LIN {X 0,Y 418.247,Z 151.387,A -85,B 0,C 180,E1 -10284.852,E2 -10284.852} C_VEL
LIN {X 0,Y 418.21,Z 151.394,A -85,B 0,C 180,E1 -10288.069,E2 -10288.069} C_VEL
LIN {X 0,Y 418.241,Z 151.389,A -85,B 0,C 180,E1 -10291.019,E2 -10291.019} C_VEL
LIN {X 0,Y 418.237,Z 151.391,A -85,B 0,C 180,E1 -10293.678,E2 -10293.678} C_VEL
LIN {X 0,Y 418.28,Z 151.466,A -85,B 0,C 180,E1 -10294.622,E2 -10294.622} C_VEL
LIN {X 0,Y 420.263,Z 161.531,A -85,B 0,C 180,E1 -10297.015,E2 -10297.015} C_VEL
LIN {X 0,Y 420.369,Z 166.895,A -85,B 0,C 180,E1 -10298.213,E2 -10298.213} C_VEL
LIN {X 0,Y 420.18,Z 169.806,A -85,B 0,C 180,E1 -10298.846,E2 -10298.846} C_VEL
LIN {X 0,Y 424.258,Z 189.635,A -85,B 0,C 180,E1 -10299.44,E2 -10299.44} C_VEL
LIN {X 0,Y 423.077,Z 277.594,A -85,B 0,C 180,E1 -10301.015,E2 -10301.015} C_VEL
LIN {X 0,Y 422.644,Z 290.834,A -85,B 0,C 180,E1 -10301.445,E2 -10301.445} C_VEL
LIN {X 0,Y 422.214,Z 302.953,A -85,B 0,C 180,E1 -10302.028,E2 -10302.028} C_VEL
LIN {X 0,Y 421.492,Z 314.996,A -85,B 0,C 180,E1 -10302.805,E2 -10302.805} C_VEL
LIN {X 0,Y 420.748,Z 326.21,A -85,B 0,C 180,E1 -10303.744,E2 -10303.744} C_VEL
LIN {X 0,Y 420.06,Z 336.204,A -85,B 0,C 180,E1 -10304.788,E2 -10304.788} C_VEL
LIN {X 0,Y 419.384,Z 345.484,A -85,B 0,C 180,E1 -10305.977,E2 -10305.977} C_VEL
LIN {X 0,Y 418.655,Z 354.531,A -85,B 0,C 180,E1 -10307.422,E2 -10307.422} C_VEL
LIN {X 0,Y 418.062,Z 362.564,A -85,B 0,C 180,E1 -10309.032,E2 -10309.032} C_VEL
LIN {X 0,Y 417.595,Z 369.077,A -85,B 0,C 180,E1 -10310.73,E2 -10310.73} C_VEL
LIN {X 0,Y 417.327,Z 373.741,A -85,B 0,C 180,E1 -10312.327,E2 -10312.327} C_VEL
LIN {X 0,Y 417.08,Z 377.245,A -85,B 0,C 180,E1 -10313.982,E2 -10313.982} C_VEL
LIN {X 0,Y 416.893,Z 379.545,A -85,B 0,C 180,E1 -10315.695,E2 -10315.695} C_VEL
LIN {X 0,Y 416.841,Z 380.55,A -85,B 0,C 180,E1 -10317.46,E2 -10317.46} C_VEL
LIN {X 0,Y 416.876,Z 380.209,A -85,B 0,C 180,E1 -10319.294,E2 -10319.294} C_VEL
LIN {X 0,Y 416.992,Z 378.31,A -85,B 0,C 180,E1 -10321.213,E2 -10321.213} C_VEL
LIN {X 0,Y 417.215,Z 375.163,A -85,B 0,C 180,E1 -10322.947,E2 -10322.947} C_VEL
LIN {X 0,Y 417.47,Z 370.897,A -85,B 0,C 180,E1 -10324.577,E2 -10324.577} C_VEL
LIN {X 0,Y 417.714,Z 365.312,A -85,B 0,C 180,E1 -10326.184,E2 -10326.184} C_VEL
LIN {X 0,Y 418.151,Z 359.125,A -85,B 0,C 180,E1 -10327.579,E2 -10327.579} C_VEL
LIN {X 0,Y 418.736,Z 350.665,A -85,B 0,C 180,E1 -10329.105,E2 -10329.105} C_VEL
LIN {X 0,Y 419.408,Z 341.621,A -85,B 0,C 180,E1 -10330.419,E2 -10330.419} C_VEL
LIN {X 0,Y 420.06,Z 331.76,A -85,B 0,C 180,E1 -10331.575,E2 -10331.575} C_VEL
LIN {X 0,Y 420.835,Z 320.491,A -85,B 0,C 180,E1 -10332.631,E2 -10332.631} C_VEL
LIN {X 0,Y 421.361,Z 310.208,A -85,B 0,C 180,E1 -10333.403,E2 -10333.403} C_VEL
LIN {X 0,Y 421.938,Z 298.072,A -85,B 0,C 180,E1 -10334.11,E2 -10334.11} C_VEL
LIN {X 0,Y 422.395,Z 285.579,A -85,B 0,C 180,E1 -10334.628,E2 -10334.628} C_VEL
LIN {X 0,Y 422.729,Z 272.036,A -85,B 0,C 180,E1 -10334.985,E2 -10334.985} C_VEL
LIN {X 0,Y 423.075,Z 245.782,A -85,B 0,C 180,E1 -10335.443,E2 -10335.443} C_VEL
LIN {X 0,Y 422.465,Z 239.979,A -85,B 0,C 180,E1 -10335.571,E2 -10335.571} C_VEL
LIN {X 0,Y 417.244,Z 221.285,A -85,B 0,C 180,E1 -10336.126,E2 -10336.126} C_VEL
LIN {X 0,Y 416.667,Z 215.482,A -85,B 0,C 180,E1 -10336.257,E2 -10336.257} C_VEL
LIN {X 0,Y 416.96,Z 190.299,A -85,B 0,C 180,E1 -10336.708,E2 -10336.708} C_VEL
LIN {X 0,Y 412.975,Z 169.781,A -85,B 0,C 180,E1 -10337.281,E2 -10337.281} C_VEL
LIN {X 0,Y 413.217,Z 162.427,A -85,B 0,C 180,E1 -10338.969,E2 -10338.969} C_VEL
LIN {X 0,Y 411.366,Z 152.245,A -85,B 0,C 180,E1 -10341.495,E2 -10341.495} C_VEL
LIN {X 0,Y 411.435,Z 152.237,A -85,B 0,C 180,E1 -10344.117,E2 -10344.117} C_VEL
LIN {X 0,Y 411.511,Z 152.224,A -85,B 0,C 180,E1 -10348.043,E2 -10348.043} C_VEL
LIN {X 0,Y 411.439,Z 152.231,A -85,B 0,C 180,E1 -10350.979,E2 -10350.979} C_VEL
LIN {X 0,Y 411.433,Z 152.232,A -85,B 0,C 180,E1 -10352.937,E2 -10352.937} C_VEL
LIN {X 0,Y 411.432,Z 152.234,A -85,B 0,C 180,E1 -10355.883,E2 -10355.883} C_VEL
LIN {X 0,Y 411.319,Z 152.246,A -85,B 0,C 180,E1 -10358.846,E2 -10358.846} C_VEL
LIN {X 0,Y 411.285,Z 152.254,A -85,B 0,C 180,E1 -10361.833,E2 -10361.833} C_VEL
LIN {X 0,Y 411.234,Z 152.256,A -85,B 0,C 180,E1 -10364.854,E2 -10364.854} C_VEL
LIN {X 0,Y 411.232,Z 152.263,A -85,B 0,C 180,E1 -10367.916,E2 -10367.916} C_VEL
LIN {X 0,Y 411.199,Z 152.26,A -85,B 0,C 180,E1 -10371.034,E2 -10371.034} C_VEL
LIN {X 0,Y 411.194,Z 152.263,A -85,B 0,C 180,E1 -10374.218,E2 -10374.218} C_VEL
LIN {X 0,Y 411.174,Z 152.268,A -85,B 0,C 180,E1 -10377.484,E2 -10377.484} C_VEL
LIN {X 0,Y 411.199,Z 152.267,A -85,B 0,C 180,E1 -10379.713,E2 -10379.713} C_VEL
LIN {X 0,Y 411.207,Z 152.262,A -85,B 0,C 180,E1 -10383.156,E2 -10383.156} C_VEL
LIN {X 0,Y 411.194,Z 152.261,A -85,B 0,C 180,E1 -10386.552,E2 -10386.552} C_VEL
LIN {X 0,Y 411.172,Z 152.267,A -85,B 0,C 180,E1 -10389.72,E2 -10389.72} C_VEL
LIN {X 0,Y 411.165,Z 152.269,A -85,B 0,C 180,E1 -10393.135,E2 -10393.135} C_VEL
LIN {X 0,Y 411.166,Z 152.265,A -85,B 0,C 180,E1 -10395.882,E2 -10395.882} C_VEL
LIN {X 0,Y 411.165,Z 152.268,A -85,B 0,C 180,E1 -10399.494,E2 -10399.494} C_VEL
LIN {X 0,Y 411.19,Z 152.261,A -85,B 0,C 180,E1 -10402.026,E2 -10402.026} C_VEL
LIN {X 0,Y 411.196,Z 152.262,A -85,B 0,C 180,E1 -10405.665,E2 -10405.665} C_VEL
LIN {X 0,Y 411.19,Z 152.266,A -85,B 0,C 180,E1 -10409.152,E2 -10409.152} C_VEL
LIN {X 0,Y 411.181,Z 152.264,A -85,B 0,C 180,E1 -10411.407,E2 -10411.407} C_VEL
LIN {X 0,Y 411.215,Z 152.264,A -85,B 0,C 180,E1 -10414.934,E2 -10414.934} C_VEL
LIN {X 0,Y 411.206,Z 152.26,A -85,B 0,C 180,E1 -10417.913,E2 -10417.913} C_VEL
LIN {X 0,Y 411.218,Z 152.261,A -85,B 0,C 180,E1 -10421.051,E2 -10421.051} C_VEL
LIN {X 0,Y 411.213,Z 152.261,A -85,B 0,C 180,E1 -10424.13,E2 -10424.13} C_VEL
LIN {X 0,Y 411.307,Z 152.248,A -85,B 0,C 180,E1 -10427.166,E2 -10427.166} C_VEL
LIN {X 0,Y 411.289,Z 152.253,A -85,B 0,C 180,E1 -10430.161,E2 -10430.161} C_VEL
LIN {X 0,Y 411.394,Z 152.236,A -85,B 0,C 180,E1 -10433.132,E2 -10433.132} C_VEL
LIN {X 0,Y 411.292,Z 152.249,A -85,B 0,C 180,E1 -10435.099,E2 -10435.099} C_VEL
LIN {X 0,Y 411.506,Z 152.227,A -85,B 0,C 180,E1 -10438.042,E2 -10438.042} C_VEL
LIN {X 0,Y 411.381,Z 152.238,A -85,B 0,C 180,E1 -10440.979,E2 -10440.979} C_VEL
LIN {X 0,Y 411.43,Z 152.232,A -85,B 0,C 180,E1 -10442.937,E2 -10442.937} C_VEL
LIN {X 0,Y 411.394,Z 152.236,A -85,B 0,C 180,E1 -10446.868,E2 -10446.868} C_VEL
LIN {X 0,Y 411.279,Z 152.256,A -85,B 0,C 180,E1 -10449.839,E2 -10449.839} C_VEL
LIN {X 0,Y 411.303,Z 152.248,A -85,B 0,C 180,E1 -10453.1,E2 -10453.1} C_VEL
LIN {X 0,Y 411.208,Z 152.259,A -85,B 0,C 180,E1 -10456.891,E2 -10456.891} C_VEL
LIN {X 0,Y 411.205,Z 152.263,A -85,B 0,C 180,E1 -10459.988,E2 -10459.988} C_VEL
LIN {X 0,Y 411.187,Z 152.264,A -85,B 0,C 180,E1 -10463.149,E2 -10463.149} C_VEL
LIN {X 0,Y 411.166,Z 152.265,A -85,B 0,C 180,E1 -10466.386,E2 -10466.386} C_VEL
LIN {X 0,Y 411.194,Z 152.265,A -85,B 0,C 180,E1 -10469.713,E2 -10469.713} C_VEL
LIN {X 0,Y 411.205,Z 152.264,A -85,B 0,C 180,E1 -10473.156,E2 -10473.156} C_VEL
LIN {X 0,Y 411.19,Z 152.262,A -85,B 0,C 180,E1 -10476.551,E2 -10476.551} C_VEL
LIN {X 0,Y 411.169,Z 152.266,A -85,B 0,C 180,E1 -10479.72,E2 -10479.72} C_VEL
LIN {X 0,Y 411.163,Z 152.272,A -85,B 0,C 180,E1 -10483.135,E2 -10483.135} C_VEL
LIN {X 0,Y 411.165,Z 152.265,A -85,B 0,C 180,E1 -10485.882,E2 -10485.882} C_VEL
LIN {X 0,Y 411.159,Z 152.267,A -85,B 0,C 180,E1 -10489.493,E2 -10489.493} C_VEL
LIN {X 0,Y 411.181,Z 152.263,A -85,B 0,C 180,E1 -10492.024,E2 -10492.024} C_VEL
LIN {X 0,Y 411.201,Z 152.264,A -85,B 0,C 180,E1 -10495.124,E2 -10495.124} C_VEL
LIN {X 0,Y 411.155,Z 152.266,A -85,B 0,C 180,E1 -10498.001,E2 -10498.001} C_VEL
LIN {X 0,Y 411.168,Z 152.269,A -85,B 0,C 180,E1 -10501.406,E2 -10501.406} C_VEL
LIN {X 0,Y 411.195,Z 152.457,A -85,B 0,C 180,E1 -10502.596,E2 -10502.596} C_VEL
LIN {X 0,Y 413.73,Z 164.949,A -85,B 0,C 180,E1 -10505.406,E2 -10505.406} C_VEL
LIN {X 0,Y 414.147,Z 168.979,A -85,B 0,C 180,E1 -10506.272,E2 -10506.272} C_VEL
LIN {X 0,Y 413.042,Z 185.931,A -85,B 0,C 180,E1 -10509.723,E2 -10509.723} C_VEL
LIN {X 0,Y 412.619,Z 190.946,A -85,B 0,C 180,E1 -10510.731,E2 -10510.731} C_VEL
LIN {X 0,Y 416.688,Z 217.687,A -85,B 0,C 180,E1 -10511.42,E2 -10511.42} C_VEL
LIN {X 0,Y 415.709,Z 299.077,A -85,B 0,C 180,E1 -10512.886,E2 -10512.886} C_VEL
LIN {X 0,Y 415.217,Z 312.276,A -85,B 0,C 180,E1 -10513.309,E2 -10513.309} C_VEL
LIN {X 0,Y 414.543,Z 325.557,A -85,B 0,C 180,E1 -10513.945,E2 -10513.945} C_VEL
LIN {X 0,Y 413.796,Z 337.523,A -85,B 0,C 180,E1 -10514.737,E2 -10514.737} C_VEL
LIN {X 0,Y 413.007,Z 349.008,A -85,B 0,C 180,E1 -10515.716,E2 -10515.716} C_VEL
LIN {X 0,Y 412.314,Z 359.362,A -85,B 0,C 180,E1 -10516.822,E2 -10516.822} C_VEL
LIN {X 0,Y 411.736,Z 367.828,A -85,B 0,C 180,E1 -10517.93,E2 -10517.93} C_VEL
LIN {X 0,Y 410.994,Z 376.995,A -85,B 0,C 180,E1 -10519.407,E2 -10519.407} C_VEL
LIN {X 0,Y 410.556,Z 384.382,A -85,B 0,C 180,E1 -10520.889,E2 -10520.889} C_VEL
LIN {X 0,Y 410.287,Z 389.386,A -85,B 0,C 180,E1 -10522.124,E2 -10522.124} C_VEL
LIN {X 0,Y 410.043,Z 394.737,A -85,B 0,C 180,E1 -10523.775,E2 -10523.775} C_VEL
LIN {X 0,Y 410.016,Z 397.958,A -85,B 0,C 180,E1 -10525.083,E2 -10525.083} C_VEL
LIN {X 0,Y 409.931,Z 399.873,A -85,B 0,C 180,E1 -10526.068,E2 -10526.068} C_VEL
LIN {X 0,Y 409.926,Z 401.342,A -85,B 0,C 180,E1 -10527.052,E2 -10527.052} C_VEL
LIN {X 0,Y 409.967,Z 402.374,A -85,B 0,C 180,E1 -10528.035,E2 -10528.035} C_VEL
LIN {X 0,Y 409.936,Z 403.011,A -85,B 0,C 180,E1 -10529.018,E2 -10529.018} C_VEL
LIN {X 0,Y 409.928,Z 403.258,A -85,B 0,C 180,E1 -10530,E2 -10530} C_VEL
LIN {X 0,Y 409.936,Z 403.087,A -85,B 0,C 180,E1 -10530.982,E2 -10530.982} C_VEL
LIN {X 0,Y 409.967,Z 402.495,A -85,B 0,C 180,E1 -10531.965,E2 -10531.965} C_VEL
LIN {X 0,Y 409.931,Z 400.127,A -85,B 0,C 180,E1 -10533.932,E2 -10533.932} C_VEL
LIN {X 0,Y 410.012,Z 397.209,A -85,B 0,C 180,E1 -10535.41,E2 -10535.41} C_VEL
LIN {X 0,Y 410.166,Z 393.255,A -85,B 0,C 180,E1 -10536.889,E2 -10536.889} C_VEL
LIN {X 0,Y 410.419,Z 388.163,A -85,B 0,C 180,E1 -10538.369,E2 -10538.369} C_VEL
LIN {X 0,Y 410.807,Z 381.768,A -85,B 0,C 180,E1 -10539.851,E2 -10539.851} C_VEL
LIN {X 0,Y 411.366,Z 373.767,A -85,B 0,C 180,E1 -10541.331,E2 -10541.331} C_VEL
LIN {X 0,Y 412.105,Z 365.627,A -85,B 0,C 180,E1 -10542.559,E2 -10542.559} C_VEL
LIN {X 0,Y 412.797,Z 355.709,A -85,B 0,C 180,E1 -10543.79,E2 -10543.79} C_VEL
LIN {X 0,Y 413.618,Z 344.608,A -85,B 0,C 180,E1 -10544.892,E2 -10544.892} C_VEL
LIN {X 0,Y 414.356,Z 333.75,A -85,B 0,C 180,E1 -10545.747,E2 -10545.747} C_VEL
LIN {X 0,Y 415.195,Z 321.802,A -85,B 0,C 180,E1 -10546.471,E2 -10546.471} C_VEL
LIN {X 0,Y 415.792,Z 308.86,A -85,B 0,C 180,E1 -10547.047,E2 -10547.047} C_VEL
LIN {X 0,Y 416.332,Z 296.141,A -85,B 0,C 180,E1 -10547.404,E2 -10547.404} C_VEL
LIN {X 0,Y 417.271,Z 216.994,A -85,B 0,C 180,E1 -10548.837,E2 -10548.837} C_VEL
LIN {X 0,Y 413.255,Z 192.477,A -85,B 0,C 180,E1 -10549.503,E2 -10549.503} C_VEL
LIN {X 0,Y 412.87,Z 190.246,A -85,B 0,C 180,E1 -10549.585,E2 -10549.585} C_VEL
LIN {X 0,Y 413.986,Z 173.404,A -85,B 0,C 180,E1 -10552.983,E2 -10552.983} C_VEL
LIN {X 0,Y 414.341,Z 168.316,A -85,B 0,C 180,E1 -10554.022,E2 -10554.022} C_VEL
LIN {X 0,Y 412.433,Z 158.109,A -85,B 0,C 180,E1 -10556.299,E2 -10556.299} C_VEL
LIN {X 0,Y 411.162,Z 152.272,A -85,B 0,C 180,E1 -10557.692,E2 -10557.692} C_VEL
LIN {X 0,Y 411.183,Z 152.269,A -85,B 0,C 180,E1 -10560.848,E2 -10560.848} C_VEL
LIN {X 0,Y 411.19,Z 152.267,A -85,B 0,C 180,E1 -10564.335,E2 -10564.335} C_VEL
LIN {X 0,Y 411.185,Z 152.266,A -85,B 0,C 180,E1 -10566.743,E2 -10566.743} C_VEL
LIN {X 0,Y 411.164,Z 152.269,A -85,B 0,C 180,E1 -10569.719,E2 -10569.719} C_VEL
LIN {X 0,Y 411.162,Z 152.274,A -85,B 0,C 180,E1 -10573.136,E2 -10573.136} C_VEL
LIN {X 0,Y 411.165,Z 152.268,A -85,B 0,C 180,E1 -10575.882,E2 -10575.882} C_VEL
LIN {X 0,Y 411.158,Z 152.265,A -85,B 0,C 180,E1 -10579.493,E2 -10579.493} C_VEL
LIN {X 0,Y 411.179,Z 152.265,A -85,B 0,C 180,E1 -10582.024,E2 -10582.024} C_VEL
LIN {X 0,Y 411.202,Z 152.264,A -85,B 0,C 180,E1 -10585.124,E2 -10585.124} C_VEL
LIN {X 0,Y 411.156,Z 152.265,A -85,B 0,C 180,E1 -10588.002,E2 -10588.002} C_VEL
LIN {X 0,Y 411.17,Z 152.262,A -85,B 0,C 180,E1 -10591.406,E2 -10591.406} C_VEL
LIN {X 0,Y 411.19,Z 152.259,A -85,B 0,C 180,E1 -10594.942,E2 -10594.942} C_VEL
LIN {X 0,Y 411.199,Z 152.262,A -85,B 0,C 180,E1 -10597.913,E2 -10597.913} C_VEL
LIN {X 0,Y 411.182,Z 152.265,A -85,B 0,C 180,E1 -10601.049,E2 -10601.049} C_VEL
LIN {X 0,Y 411.199,Z 152.259,A -85,B 0,C 180,E1 -10604.129,E2 -10604.129} C_VEL
LIN {X 0,Y 411.299,Z 152.248,A -85,B 0,C 180,E1 -10607.166,E2 -10607.166} C_VEL
LIN {X 0,Y 411.277,Z 152.25,A -85,B 0,C 180,E1 -10610.161,E2 -10610.161} C_VEL
LIN {X 0,Y 411.392,Z 152.23,A -85,B 0,C 180,E1 -10613.132,E2 -10613.132} C_VEL
LIN {X 0,Y 411.286,Z 152.249,A -85,B 0,C 180,E1 -10615.099,E2 -10615.099} C_VEL
LIN {X 0,Y 411.506,Z 152.22,A -85,B 0,C 180,E1 -10618.043,E2 -10618.043} C_VEL
LIN {X 0,Y 411.381,Z 152.236,A -85,B 0,C 180,E1 -10620.979,E2 -10620.979} C_VEL
LIN {X 0,Y 411.43,Z 152.232,A -85,B 0,C 180,E1 -10622.938,E2 -10622.938} C_VEL
LIN {X 0,Y 411.394,Z 152.237,A -85,B 0,C 180,E1 -10626.868,E2 -10626.868} C_VEL
LIN {X 0,Y 411.28,Z 152.252,A -85,B 0,C 180,E1 -10629.839,E2 -10629.839} C_VEL
LIN {X 0,Y 411.309,Z 152.246,A -85,B 0,C 180,E1 -10633.103,E2 -10633.103} C_VEL
LIN {X 0,Y 411.211,Z 152.261,A -85,B 0,C 180,E1 -10636.891,E2 -10636.891} C_VEL
LIN {X 0,Y 411.207,Z 152.263,A -85,B 0,C 180,E1 -10639.988,E2 -10639.988} C_VEL
LIN {X 0,Y 411.192,Z 152.265,A -85,B 0,C 180,E1 -10643.148,E2 -10643.148} C_VEL
LIN {X 0,Y 411.178,Z 152.269,A -85,B 0,C 180,E1 -10646.385,E2 -10646.385} C_VEL
LIN {X 0,Y 411.198,Z 152.267,A -85,B 0,C 180,E1 -10649.713,E2 -10649.713} C_VEL
LIN {X 0,Y 411.208,Z 152.265,A -85,B 0,C 180,E1 -10653.156,E2 -10653.156} C_VEL
LIN {X 0,Y 411.217,Z 152.351,A -85,B 0,C 180,E1 -10654.333,E2 -10654.333} C_VEL
LIN {X 0,Y 413.378,Z 163.207,A -85,B 0,C 180,E1 -10656.958,E2 -10656.958} C_VEL
LIN {X 0,Y 413.45,Z 168.137,A -85,B 0,C 180,E1 -10658.077,E2 -10658.077} C_VEL
LIN {X 0,Y 413.332,Z 170.075,A -85,B 0,C 180,E1 -10658.506,E2 -10658.506} C_VEL
LIN {X 0,Y 417.683,Z 191.349,A -85,B 0,C 180,E1 -10659.142,E2 -10659.142} C_VEL
LIN {X 0,Y 416.348,Z 277.624,A -85,B 0,C 180,E1 -10660.707,E2 -10660.707} C_VEL
LIN {X 0,Y 415.892,Z 291.111,A -85,B 0,C 180,E1 -10661.151,E2 -10661.151} C_VEL
LIN {X 0,Y 415.423,Z 303.31,A -85,B 0,C 180,E1 -10661.749,E2 -10661.749} C_VEL
LIN {X 0,Y 414.653,Z 315.611,A -85,B 0,C 180,E1 -10662.563,E2 -10662.563} C_VEL
LIN {X 0,Y 413.844,Z 327.228,A -85,B 0,C 180,E1 -10663.564,E2 -10663.564} C_VEL
LIN {X 0,Y 413.044,Z 337.978,A -85,B 0,C 180,E1 -10664.733,E2 -10664.733} C_VEL
LIN {X 0,Y 412.299,Z 347.356,A -85,B 0,C 180,E1 -10666.009,E2 -10666.009} C_VEL
LIN {X 0,Y 411.681,Z 354.747,A -85,B 0,C 180,E1 -10667.229,E2 -10667.229} C_VEL
LIN {X 0,Y 411.07,Z 362.421,A -85,B 0,C 180,E1 -10668.787,E2 -10668.787} C_VEL
LIN {X 0,Y 410.601,Z 368.581,A -85,B 0,C 180,E1 -10670.375,E2 -10670.375} C_VEL
LIN {X 0,Y 410.279,Z 373.398,A -85,B 0,C 180,E1 -10671.997,E2 -10671.997} C_VEL
LIN {X 0,Y 410.033,Z 377.03,A -85,B 0,C 180,E1 -10673.667,E2 -10673.667} C_VEL
LIN {X 0,Y 409.804,Z 379.64,A -85,B 0,C 180,E1 -10675.532,E2 -10675.532} C_VEL
LIN {X 0,Y 409.739,Z 380.707,A -85,B 0,C 180,E1 -10677.19,E2 -10677.19} C_VEL
LIN {X 0,Y 409.765,Z 380.532,A -85,B 0,C 180,E1 -10679.045,E2 -10679.045} C_VEL
LIN {X 0,Y 409.829,Z 379.751,A -85,B 0,C 180,E1 -10680.178,E2 -10680.178} C_VEL
LIN {X 0,Y 409.903,Z 378.415,A -85,B 0,C 180,E1 -10681.309,E2 -10681.309} C_VEL
LIN {X 0,Y 410.129,Z 375.365,A -85,B 0,C 180,E1 -10683.009,E2 -10683.009} C_VEL
LIN {X 0,Y 410.41,Z 371.144,A -85,B 0,C 180,E1 -10684.652,E2 -10684.652} C_VEL
LIN {X 0,Y 410.677,Z 365.574,A -85,B 0,C 180,E1 -10686.286,E2 -10686.286} C_VEL
LIN {X 0,Y 411.18,Z 358.374,A -85,B 0,C 180,E1 -10687.912,E2 -10687.912} C_VEL
LIN {X 0,Y 411.795,Z 349.969,A -85,B 0,C 180,E1 -10689.421,E2 -10689.421} C_VEL
LIN {X 0,Y 412.499,Z 340.937,A -85,B 0,C 180,E1 -10690.725,E2 -10690.725} C_VEL
LIN {X 0,Y 413.23,Z 330.683,A -85,B 0,C 180,E1 -10691.917,E2 -10691.917} C_VEL
LIN {X 0,Y 414.005,Z 319.36,A -85,B 0,C 180,E1 -10692.972,E2 -10692.972} C_VEL
LIN {X 0,Y 414.639,Z 307.674,A -85,B 0,C 180,E1 -10693.823,E2 -10693.823} C_VEL
LIN {X 0,Y 415.16,Z 295.909,A -85,B 0,C 180,E1 -10694.473,E2 -10694.473} C_VEL
LIN {X 0,Y 415.664,Z 282.878,A -85,B 0,C 180,E1 -10694.984,E2 -10694.984} C_VEL
LIN {X 0,Y 415.96,Z 269.747,A -85,B 0,C 180,E1 -10695.297,E2 -10695.297} C_VEL
LIN {X 0,Y 416.667,Z 215.482,A -85,B 0,C 180,E1 -10696.257,E2 -10696.257} C_VEL
LIN {X 0,Y 416.139,Z 209.665,A -85,B 0,C 180,E1 -10696.387,E2 -10696.387} C_VEL
LIN {X 0,Y 413.596,Z 200.312,A -85,B 0,C 180,E1 -10696.671,E2 -10696.671} C_VEL
LIN {X 0,Y 411.065,Z 192.914,A -85,B 0,C 180,E1 -10696.922,E2 -10696.922} C_VEL
LIN {X 0,Y 409.064,Z 185.346,A -85,B 0,C 180,E1 -10697.155,E2 -10697.155} C_VEL
LIN {X 0,Y 406.073,Z 169.943,A -85,B 0,C 180,E1 -10697.601,E2 -10697.601} C_VEL
LIN {X 0,Y 406.261,Z 163.82,A -85,B 0,C 180,E1 -10699.03,E2 -10699.03} C_VEL
LIN {X 0,Y 404.318,Z 153.123,A -85,B 0,C 180,E1 -10701.724,E2 -10701.724} C_VEL
LIN {X 0,Y 404.382,Z 153.116,A -85,B 0,C 180,E1 -10704.014,E2 -10704.014} C_VEL
LIN {X 0,Y 404.48,Z 153.1,A -85,B 0,C 180,E1 -10708.008,E2 -10708.008} C_VEL
LIN {X 0,Y 404.404,Z 153.108,A -85,B 0,C 180,E1 -10710.996,E2 -10710.996} C_VEL
LIN {X 0,Y 404.392,Z 153.109,A -85,B 0,C 180,E1 -10712.989,E2 -10712.989} C_VEL
LIN {X 0,Y 404.38,Z 153.114,A -85,B 0,C 180,E1 -10715.986,E2 -10715.986} C_VEL
LIN {X 0,Y 404.267,Z 153.124,A -85,B 0,C 180,E1 -10719.002,E2 -10719.002} C_VEL
LIN {X 0,Y 404.258,Z 153.132,A -85,B 0,C 180,E1 -10722.042,E2 -10722.042} C_VEL
LIN {X 0,Y 404.179,Z 153.135,A -85,B 0,C 180,E1 -10725.119,E2 -10725.119} C_VEL
LIN {X 0,Y 404.196,Z 153.136,A -85,B 0,C 180,E1 -10728.239,E2 -10728.239} C_VEL
LIN {X 0,Y 404.141,Z 153.142,A -85,B 0,C 180,E1 -10731.419,E2 -10731.419} C_VEL
LIN {X 0,Y 404.15,Z 153.138,A -85,B 0,C 180,E1 -10734.668,E2 -10734.668} C_VEL
LIN {X 0,Y 404.118,Z 153.146,A -85,B 0,C 180,E1 -10738.006,E2 -10738.006} C_VEL
LIN {X 0,Y 404.146,Z 153.14,A -85,B 0,C 180,E1 -10740.285,E2 -10740.285} C_VEL
LIN {X 0,Y 404.14,Z 153.144,A -85,B 0,C 180,E1 -10743.813,E2 -10743.813} C_VEL
LIN {X 0,Y 404.137,Z 153.141,A -85,B 0,C 180,E1 -10746.875,E2 -10746.875} C_VEL
LIN {X 0,Y 404.119,Z 153.143,A -85,B 0,C 180,E1 -10750.075,E2 -10750.075} C_VEL
LIN {X 0,Y 404.144,Z 153.143,A -85,B 0,C 180,E1 -10753.082,E2 -10753.082} C_VEL
LIN {X 0,Y 404.123,Z 153.143,A -85,B 0,C 180,E1 -10755.922,E2 -10755.922} C_VEL
LIN {X 0,Y 404.106,Z 153.145,A -85,B 0,C 180,E1 -10758.633,E2 -10758.633} C_VEL
LIN {X 0,Y 404.145,Z 153.142,A -85,B 0,C 180,E1 -10761.494,E2 -10761.494} C_VEL
LIN {X 0,Y 404.177,Z 153.141,A -85,B 0,C 180,E1 -10764.983,E2 -10764.983} C_VEL
LIN {X 0,Y 404.14,Z 153.141,A -85,B 0,C 180,E1 -10768.443,E2 -10768.443} C_VEL
LIN {X 0,Y 404.154,Z 153.145,A -85,B 0,C 180,E1 -10770.863,E2 -10770.863} C_VEL
LIN {X 0,Y 404.143,Z 153.141,A -85,B 0,C 180,E1 -10774.231,E2 -10774.231} C_VEL
LIN {X 0,Y 404.169,Z 153.136,A -85,B 0,C 180,E1 -10777.508,E2 -10777.508} C_VEL
LIN {X 0,Y 404.163,Z 153.143,A -85,B 0,C 180,E1 -10780.707,E2 -10780.707} C_VEL
LIN {X 0,Y 404.184,Z 153.135,A -85,B 0,C 180,E1 -10783.846,E2 -10783.846} C_VEL
LIN {X 0,Y 404.287,Z 153.124,A -85,B 0,C 180,E1 -10786.939,E2 -10786.939} C_VEL
LIN {X 0,Y 404.256,Z 153.128,A -85,B 0,C 180,E1 -10789.988,E2 -10789.988} C_VEL
LIN {X 0,Y 404.344,Z 153.115,A -85,B 0,C 180,E1 -10793.012,E2 -10793.012} C_VEL
LIN {X 0,Y 404.263,Z 153.125,A -85,B 0,C 180,E1 -10795.013,E2 -10795.013} C_VEL
LIN {X 0,Y 404.475,Z 153.102,A -85,B 0,C 180,E1 -10798.008,E2 -10798.008} C_VEL
LIN {X 0,Y 404.352,Z 153.114,A -85,B 0,C 180,E1 -10800.996,E2 -10800.996} C_VEL
LIN {X 0,Y 404.389,Z 153.109,A -85,B 0,C 180,E1 -10802.989,E2 -10802.989} C_VEL
LIN {X 0,Y 404.37,Z 153.117,A -85,B 0,C 180,E1 -10805.986,E2 -10805.986} C_VEL
LIN {X 0,Y 404.259,Z 153.125,A -85,B 0,C 180,E1 -10809.002,E2 -10809.002} C_VEL
LIN {X 0,Y 404.249,Z 153.131,A -85,B 0,C 180,E1 -10812.042,E2 -10812.042} C_VEL
LIN {X 0,Y 404.16,Z 153.138,A -85,B 0,C 180,E1 -10815.12,E2 -10815.12} C_VEL
LIN {X 0,Y 404.13,Z 153.143,A -85,B 0,C 180,E1 -10818.242,E2 -10818.242} C_VEL
LIN {X 0,Y 404.129,Z 153.145,A -85,B 0,C 180,E1 -10821.42,E2 -10821.42} C_VEL
LIN {X 0,Y 404.136,Z 153.14,A -85,B 0,C 180,E1 -10824.668,E2 -10824.668} C_VEL
LIN {X 0,Y 404.101,Z 153.146,A -85,B 0,C 180,E1 -10828.007,E2 -10828.007} C_VEL
LIN {X 0,Y 404.141,Z 153.14,A -85,B 0,C 180,E1 -10830.286,E2 -10830.286} C_VEL
LIN {X 0,Y 404.138,Z 153.142,A -85,B 0,C 180,E1 -10833.813,E2 -10833.813} C_VEL
LIN {X 0,Y 404.133,Z 153.143,A -85,B 0,C 180,E1 -10836.874,E2 -10836.874} C_VEL
LIN {X 0,Y 404.119,Z 153.142,A -85,B 0,C 180,E1 -10840.075,E2 -10840.075} C_VEL
LIN {X 0,Y 404.143,Z 153.146,A -85,B 0,C 180,E1 -10843.082,E2 -10843.082} C_VEL
LIN {X 0,Y 404.122,Z 153.142,A -85,B 0,C 180,E1 -10845.922,E2 -10845.922} C_VEL
LIN {X 0,Y 404.102,Z 153.147,A -85,B 0,C 180,E1 -10848.632,E2 -10848.632} C_VEL
LIN {X 0,Y 404.138,Z 153.141,A -85,B 0,C 180,E1 -10851.495,E2 -10851.495} C_VEL
LIN {X 0,Y 404.172,Z 153.141,A -85,B 0,C 180,E1 -10854.982,E2 -10854.982} C_VEL
LIN {X 0,Y 404.132,Z 153.144,A -85,B 0,C 180,E1 -10858.444,E2 -10858.444} C_VEL
LIN {X 0,Y 404.148,Z 153.145,A -85,B 0,C 180,E1 -10860.862,E2 -10860.862} C_VEL
LIN {X 0,Y 404.169,Z 153.289,A -85,B 0,C 180,E1 -10862.333,E2 -10862.333} C_VEL
LIN {X 0,Y 406.703,Z 165.919,A -85,B 0,C 180,E1 -10865.225,E2 -10865.225} C_VEL
LIN {X 0,Y 407.202,Z 170.22,A -85,B 0,C 180,E1 -10866.169,E2 -10866.169} C_VEL
LIN {X 0,Y 406.019,Z 187.492,A -85,B 0,C 180,E1 -10869.745,E2 -10869.745} C_VEL
LIN {X 0,Y 405.704,Z 190.807,A -85,B 0,C 180,E1 -10870.422,E2 -10870.422} C_VEL
LIN {X 0,Y 409.925,Z 218.175,A -85,B 0,C 180,E1 -10871.133,E2 -10871.133} C_VEL
LIN {X 0,Y 408.886,Z 299.259,A -85,B 0,C 180,E1 -10872.624,E2 -10872.624} C_VEL
LIN {X 0,Y 408.343,Z 313.089,A -85,B 0,C 180,E1 -10873.084,E2 -10873.084} C_VEL
LIN {X 0,Y 407.649,Z 326.057,A -85,B 0,C 180,E1 -10873.73,E2 -10873.73} C_VEL
LIN {X 0,Y 406.817,Z 338.65,A -85,B 0,C 180,E1 -10874.597,E2 -10874.597} C_VEL
LIN {X 0,Y 406.032,Z 349.897,A -85,B 0,C 180,E1 -10875.593,E2 -10875.593} C_VEL
LIN {X 0,Y 405.268,Z 360.185,A -85,B 0,C 180,E1 -10876.739,E2 -10876.739} C_VEL
LIN {X 0,Y 404.621,Z 369.147,A -85,B 0,C 180,E1 -10877.969,E2 -10877.969} C_VEL
LIN {X 0,Y 403.905,Z 378.058,A -85,B 0,C 180,E1 -10879.473,E2 -10879.473} C_VEL
LIN {X 0,Y 403.473,Z 385.201,A -85,B 0,C 180,E1 -10880.981,E2 -10880.981} C_VEL
LIN {X 0,Y 403.137,Z 390.89,A -85,B 0,C 180,E1 -10882.487,E2 -10882.487} C_VEL
LIN {X 0,Y 402.938,Z 395.363,A -85,B 0,C 180,E1 -10883.993,E2 -10883.993} C_VEL
LIN {X 0,Y 402.928,Z 397.723,A -85,B 0,C 180,E1 -10884.997,E2 -10884.997} C_VEL
LIN {X 0,Y 402.851,Z 399.646,A -85,B 0,C 180,E1 -10885.998,E2 -10885.998} C_VEL
LIN {X 0,Y 402.825,Z 401.127,A -85,B 0,C 180,E1 -10887,E2 -10887} C_VEL
LIN {X 0,Y 402.865,Z 402.165,A -85,B 0,C 180,E1 -10888.001,E2 -10888.001} C_VEL
LIN {X 0,Y 402.863,Z 402.808,A -85,B 0,C 180,E1 -10889,E2 -10889} C_VEL
LIN {X 0,Y 402.853,Z 403.061,A -85,B 0,C 180,E1 -10890,E2 -10890} C_VEL
LIN {X 0,Y 402.863,Z 402.9,A -85,B 0,C 180,E1 -10891,E2 -10891} C_VEL
LIN {X 0,Y 402.864,Z 402.312,A -85,B 0,C 180,E1 -10892,E2 -10892} C_VEL
LIN {X 0,Y 402.851,Z 399.953,A -85,B 0,C 180,E1 -10894.002,E2 -10894.002} C_VEL
LIN {X 0,Y 402.909,Z 397.044,A -85,B 0,C 180,E1 -10895.505,E2 -10895.505} C_VEL
LIN {X 0,Y 403.08,Z 393.098,A -85,B 0,C 180,E1 -10897.011,E2 -10897.011} C_VEL
LIN {X 0,Y 403.36,Z 388.016,A -85,B 0,C 180,E1 -10898.517,E2 -10898.517} C_VEL
LIN {X 0,Y 403.802,Z 381.643,A -85,B 0,C 180,E1 -10900.023,E2 -10900.023} C_VEL
LIN {X 0,Y 404.385,Z 373.668,A -85,B 0,C 180,E1 -10901.529,E2 -10901.529} C_VEL
LIN {X 0,Y 405.159,Z 365.557,A -85,B 0,C 180,E1 -10902.778,E2 -10902.778} C_VEL
LIN {X 0,Y 405.873,Z 355.673,A -85,B 0,C 180,E1 -10904.03,E2 -10904.03} C_VEL
LIN {X 0,Y 406.764,Z 344.626,A -85,B 0,C 180,E1 -10905.149,E2 -10905.149} C_VEL
LIN {X 0,Y 407.539,Z 333.819,A -85,B 0,C 180,E1 -10906.017,E2 -10906.017} C_VEL
LIN {X 0,Y 408.412,Z 321.946,A -85,B 0,C 180,E1 -10906.753,E2 -10906.753} C_VEL
LIN {X 0,Y 409.037,Z 309.184,A -85,B 0,C 180,E1 -10907.338,E2 -10907.338} C_VEL
LIN {X 0,Y 409.602,Z 295.396,A -85,B 0,C 180,E1 -10907.732,E2 -10907.732} C_VEL
LIN {X 0,Y 410.506,Z 216.867,A -85,B 0,C 180,E1 -10909.182,E2 -10909.182} C_VEL
LIN {X 0,Y 406.354,Z 192.13,A -85,B 0,C 180,E1 -10909.88,E2 -10909.88} C_VEL
LIN {X 0,Y 406.022,Z 190,A -85,B 0,C 180,E1 -10909.964,E2 -10909.964} C_VEL
LIN {X 0,Y 407.356,Z 171.699,A -85,B 0,C 180,E1 -10913.727,E2 -10913.727} C_VEL
LIN {X 0,Y 407.24,Z 168.248,A -85,B 0,C 180,E1 -10914.468,E2 -10914.468} C_VEL
LIN {X 0,Y 405.197,Z 158.058,A -85,B 0,C 180,E1 -10916.806,E2 -10916.806} C_VEL
LIN {X 0,Y 404.118,Z 153.152,A -85,B 0,C 180,E1 -10918.006,E2 -10918.006} C_VEL
LIN {X 0,Y 404.14,Z 153.148,A -85,B 0,C 180,E1 -10920.286,E2 -10920.286} C_VEL
LIN {X 0,Y 404.137,Z 153.147,A -85,B 0,C 180,E1 -10923.813,E2 -10923.813} C_VEL
LIN {X 0,Y 404.131,Z 153.145,A -85,B 0,C 180,E1 -10926.874,E2 -10926.874} C_VEL
LIN {X 0,Y 404.119,Z 153.146,A -85,B 0,C 180,E1 -10930.075,E2 -10930.075} C_VEL
LIN {X 0,Y 404.142,Z 153.149,A -85,B 0,C 180,E1 -10933.082,E2 -10933.082} C_VEL
LIN {X 0,Y 404.122,Z 153.145,A -85,B 0,C 180,E1 -10935.922,E2 -10935.922} C_VEL
LIN {X 0,Y 404.102,Z 153.15,A -85,B 0,C 180,E1 -10938.633,E2 -10938.633} C_VEL
LIN {X 0,Y 404.135,Z 153.143,A -85,B 0,C 180,E1 -10941.496,E2 -10941.496} C_VEL
LIN {X 0,Y 404.173,Z 153.141,A -85,B 0,C 180,E1 -10944.983,E2 -10944.983} C_VEL
LIN {X 0,Y 404.133,Z 153.143,A -85,B 0,C 180,E1 -10948.444,E2 -10948.444} C_VEL
LIN {X 0,Y 404.149,Z 153.137,A -85,B 0,C 180,E1 -10950.862,E2 -10950.862} C_VEL
LIN {X 0,Y 404.154,Z 153.136,A -85,B 0,C 180,E1 -10954.724,E2 -10954.724} C_VEL
LIN {X 0,Y 404.165,Z 153.137,A -85,B 0,C 180,E1 -10957.508,E2 -10957.508} C_VEL
LIN {X 0,Y 404.135,Z 153.143,A -85,B 0,C 180,E1 -10960.706,E2 -10960.706} C_VEL
LIN {X 0,Y 404.174,Z 153.134,A -85,B 0,C 180,E1 -10963.846,E2 -10963.846} C_VEL
LIN {X 0,Y 404.268,Z 153.125,A -85,B 0,C 180,E1 -10966.938,E2 -10966.938} C_VEL
LIN {X 0,Y 404.245,Z 153.124,A -85,B 0,C 180,E1 -10969.988,E2 -10969.988} C_VEL
LIN {X 0,Y 404.342,Z 153.108,A -85,B 0,C 180,E1 -10973.012,E2 -10973.012} C_VEL
LIN {X 0,Y 404.258,Z 153.124,A -85,B 0,C 180,E1 -10975.013,E2 -10975.013} C_VEL
LIN {X 0,Y 404.474,Z 153.095,A -85,B 0,C 180,E1 -10978.009,E2 -10978.009} C_VEL
LIN {X 0,Y 404.351,Z 153.111,A -85,B 0,C 180,E1 -10980.996,E2 -10980.996} C_VEL
LIN {X 0,Y 404.363,Z 153.112,A -85,B 0,C 180,E1 -10982.989,E2 -10982.989} C_VEL
LIN {X 0,Y 404.342,Z 153.113,A -85,B 0,C 180,E1 -10986.485,E2 -10986.485} C_VEL
LIN {X 0,Y 404.26,Z 153.123,A -85,B 0,C 180,E1 -10989.002,E2 -10989.002} C_VEL
LIN {X 0,Y 404.253,Z 153.128,A -85,B 0,C 180,E1 -10992.042,E2 -10992.042} C_VEL
LIN {X 0,Y 404.178,Z 153.137,A -85,B 0,C 180,E1 -10995.119,E2 -10995.119} C_VEL
LIN {X 0,Y 404.139,Z 153.143,A -85,B 0,C 180,E1 -10998.242,E2 -10998.242} C_VEL
LIN {X 0,Y 404.135,Z 153.145,A -85,B 0,C 180,E1 -11001.42,E2 -11001.42} C_VEL
LIN {X 0,Y 404.152,Z 153.143,A -85,B 0,C 180,E1 -11004.667,E2 -11004.667} C_VEL
LIN {X 0,Y 404.106,Z 153.152,A -85,B 0,C 180,E1 -11008.007,E2 -11008.007} C_VEL
LIN {X 0,Y 404.145,Z 153.144,A -85,B 0,C 180,E1 -11010.285,E2 -11010.285} C_VEL
LIN {X 0,Y 404.201,Z 153.279,A -85,B 0,C 180,E1 -11014.032,E2 -11014.032} C_VEL
LIN {X 0,Y 406.319,Z 163.813,A -85,B 0,C 180,E1 -11016.637,E2 -11016.637} C_VEL
LIN {X 0,Y 406.662,Z 166.791,A -85,B 0,C 180,E1 -11017.346,E2 -11017.346} C_VEL
LIN {X 0,Y 406.5,Z 170.434,A -85,B 0,C 180,E1 -11018.145,E2 -11018.145} C_VEL
LIN {X 0,Y 410.928,Z 191.578,A -85,B 0,C 180,E1 -11018.797,E2 -11018.797} C_VEL
LIN {X 0,Y 409.607,Z 278.396,A -85,B 0,C 180,E1 -11020.409,E2 -11020.409} C_VEL
LIN {X 0,Y 409.136,Z 292.217,A -85,B 0,C 180,E1 -11020.883,E2 -11020.883} C_VEL
LIN {X 0,Y 408.573,Z 305.291,A -85,B 0,C 180,E1 -11021.56,E2 -11021.56} C_VEL
LIN {X 0,Y 407.725,Z 317.522,A -85,B 0,C 180,E1 -11022.413,E2 -11022.413} C_VEL
LIN {X 0,Y 406.992,Z 327.769,A -85,B 0,C 180,E1 -11023.329,E2 -11023.329} C_VEL
LIN {X 0,Y 406.169,Z 337.981,A -85,B 0,C 180,E1 -11024.458,E2 -11024.458} C_VEL
LIN {X 0,Y 405.379,Z 347.513,A -85,B 0,C 180,E1 -11025.773,E2 -11025.773} C_VEL
LIN {X 0,Y 404.547,Z 356.71,A -85,B 0,C 180,E1 -11027.349,E2 -11027.349} C_VEL
LIN {X 0,Y 403.951,Z 364.022,A -85,B 0,C 180,E1 -11028.945,E2 -11028.945} C_VEL
LIN {X 0,Y 403.495,Z 369.931,A -85,B 0,C 180,E1 -11030.585,E2 -11030.585} C_VEL
LIN {X 0,Y 403.153,Z 374.88,A -85,B 0,C 180,E1 -11032.4,E2 -11032.4} C_VEL
LIN {X 0,Y 402.962,Z 377.326,A -85,B 0,C 180,E1 -11033.63,E2 -11033.63} C_VEL
LIN {X 0,Y 402.741,Z 379.427,A -85,B 0,C 180,E1 -11035.102,E2 -11035.102} C_VEL
LIN {X 0,Y 402.663,Z 380.797,A -85,B 0,C 180,E1 -11036.907,E2 -11036.907} C_VEL
LIN {X 0,Y 402.648,Z 380.852,A -85,B 0,C 180,E1 -11038.79,E2 -11038.79} C_VEL
LIN {X 0,Y 402.768,Z 379.359,A -85,B 0,C 180,E1 -11040.752,E2 -11040.752} C_VEL
LIN {X 0,Y 402.868,Z 377.798,A -85,B 0,C 180,E1 -11041.9,E2 -11041.9} C_VEL
LIN {X 0,Y 403.143,Z 374.377,A -85,B 0,C 180,E1 -11043.606,E2 -11043.606} C_VEL
LIN {X 0,Y 403.414,Z 369.69,A -85,B 0,C 180,E1 -11045.284,E2 -11045.284} C_VEL
LIN {X 0,Y 403.781,Z 363.924,A -85,B 0,C 180,E1 -11046.869,E2 -11046.869} C_VEL
LIN {X 0,Y 404.234,Z 357.316,A -85,B 0,C 180,E1 -11048.318,E2 -11048.318} C_VEL
LIN {X 0,Y 404.874,Z 349.638,A -85,B 0,C 180,E1 -11049.685,E2 -11049.685} C_VEL
LIN {X 0,Y 405.605,Z 340.215,A -85,B 0,C 180,E1 -11051.041,E2 -11051.041} C_VEL
LIN {X 0,Y 406.331,Z 330.28,A -85,B 0,C 180,E1 -11052.2,E2 -11052.2} C_VEL
LIN {X 0,Y 407.1,Z 319.751,A -85,B 0,C 180,E1 -11053.192,E2 -11053.192} C_VEL
LIN {X 0,Y 407.792,Z 307.683,A -85,B 0,C 180,E1 -11054.084,E2 -11054.084} C_VEL
LIN {X 0,Y 408.356,Z 295.077,A -85,B 0,C 180,E1 -11054.783,E2 -11054.783} C_VEL
LIN {X 0,Y 408.873,Z 282.217,A -85,B 0,C 180,E1 -11055.281,E2 -11055.281} C_VEL
LIN {X 0,Y 409.175,Z 267.79,A -85,B 0,C 180,E1 -11055.61,E2 -11055.61} C_VEL
LIN {X 0,Y 410.217,Z 191.382,A -85,B 0,C 180,E1 -11056.989,E2 -11056.989} C_VEL
LIN {X 0,Y 409.064,Z 185.346,A -85,B 0,C 180,E1 -11057.155,E2 -11057.155} C_VEL
LIN {X 0,Y 407.507,Z 180.011,A -85,B 0,C 180,E1 -11057.381,E2 -11057.381} C_VEL
LIN {X 0,Y 405.281,Z 175.244,A -85,B 0,C 180,E1 -11057.733,E2 -11057.733} C_VEL
LIN {X 0,Y 402.087,Z 169.715,A -85,B 0,C 180,E1 -11058.371,E2 -11058.371} C_VEL
LIN {X 0,Y 400.068,Z 166.114,A -85,B 0,C 180,E1 -11058.966,E2 -11058.966} C_VEL
LIN {X 0,Y 398.903,Z 162.979,A -85,B 0,C 180,E1 -11059.652,E2 -11059.652} C_VEL
LIN {X 0,Y 397.299,Z 153.995,A -85,B 0,C 180,E1 -11061.964,E2 -11061.964} C_VEL
LIN {X 0,Y 397.242,Z 154.001,A -85,B 0,C 180,E1 -11064.925,E2 -11064.925} C_VEL
LIN {X 0,Y 397.449,Z 153.975,A -85,B 0,C 180,E1 -11067.973,E2 -11067.973} C_VEL
LIN {X 0,Y 397.369,Z 153.984,A -85,B 0,C 180,E1 -11071.013,E2 -11071.013} C_VEL
LIN {X 0,Y 397.327,Z 153.989,A -85,B 0,C 180,E1 -11073.042,E2 -11073.042} C_VEL
LIN {X 0,Y 397.331,Z 153.993,A -85,B 0,C 180,E1 -11076.092,E2 -11076.092} C_VEL
LIN {X 0,Y 397.237,Z 154,A -85,B 0,C 180,E1 -11079.162,E2 -11079.162} C_VEL
LIN {X 0,Y 397.221,Z 154.006,A -85,B 0,C 180,E1 -11082.258,E2 -11082.258} C_VEL
LIN {X 0,Y 397.127,Z 154.014,A -85,B 0,C 180,E1 -11085.394,E2 -11085.394} C_VEL
LIN {X 0,Y 397.153,Z 154.011,A -85,B 0,C 180,E1 -11088.574,E2 -11088.574} C_VEL
LIN {X 0,Y 397.098,Z 154.024,A -85,B 0,C 180,E1 -11091.819,E2 -11091.819} C_VEL
LIN {X 0,Y 397.098,Z 154.018,A -85,B 0,C 180,E1 -11095.136,E2 -11095.136} C_VEL
LIN {X 0,Y 397.072,Z 154.02,A -85,B 0,C 180,E1 -11098.548,E2 -11098.548} C_VEL
LIN {X 0,Y 397.083,Z 154.023,A -85,B 0,C 180,E1 -11101.836,E2 -11101.836} C_VEL
LIN {X 0,Y 397.122,Z 154.014,A -85,B 0,C 180,E1 -11104.494,E2 -11104.494} C_VEL
LIN {X 0,Y 397.095,Z 154.018,A -85,B 0,C 180,E1 -11108.276,E2 -11108.276} C_VEL
LIN {X 0,Y 397.054,Z 154.023,A -85,B 0,C 180,E1 -11111.977,E2 -11111.977} C_VEL
LIN {X 0,Y 397.088,Z 154.023,A -85,B 0,C 180,E1 -11115.069,E2 -11115.069} C_VEL
LIN {X 0,Y 397.054,Z 154.023,A -85,B 0,C 180,E1 -11118.024,E2 -11118.024} C_VEL
LIN {X 0,Y 397.096,Z 154.018,A -85,B 0,C 180,E1 -11121.724,E2 -11121.724} C_VEL
LIN {X 0,Y 397.12,Z 154.016,A -85,B 0,C 180,E1 -11125.506,E2 -11125.506} C_VEL
LIN {X 0,Y 397.079,Z 154.024,A -85,B 0,C 180,E1 -11129.117,E2 -11129.117} C_VEL
LIN {X 0,Y 397.094,Z 154.021,A -85,B 0,C 180,E1 -11132.602,E2 -11132.602} C_VEL
LIN {X 0,Y 397.115,Z 154.015,A -85,B 0,C 180,E1 -11135.98,E2 -11135.98} C_VEL
LIN {X 0,Y 397.142,Z 154.011,A -85,B 0,C 180,E1 -11139.705,E2 -11139.705} C_VEL
LIN {X 0,Y 397.157,Z 154.014,A -85,B 0,C 180,E1 -11142.859,E2 -11142.859} C_VEL
LIN {X 0,Y 397.233,Z 154.005,A -85,B 0,C 180,E1 -11146.703,E2 -11146.703} C_VEL
LIN {X 0,Y 397.216,Z 154.003,A -85,B 0,C 180,E1 -11149.809,E2 -11149.809} C_VEL
LIN {X 0,Y 397.297,Z 153.994,A -85,B 0,C 180,E1 -11152.887,E2 -11152.887} C_VEL
LIN {X 0,Y 397.235,Z 154.001,A -85,B 0,C 180,E1 -11154.925,E2 -11154.925} C_VEL
LIN {X 0,Y 397.443,Z 153.978,A -85,B 0,C 180,E1 -11157.973,E2 -11157.973} C_VEL
LIN {X 0,Y 397.443,Z 153.98,A -85,B 0,C 180,E1 -11162.027,E2 -11162.027} C_VEL
LIN {X 0,Y 397.323,Z 153.995,A -85,B 0,C 180,E1 -11166.092,E2 -11166.092} C_VEL
LIN {X 0,Y 397.23,Z 154.001,A -85,B 0,C 180,E1 -11169.162,E2 -11169.162} C_VEL
LIN {X 0,Y 397.211,Z 154.006,A -85,B 0,C 180,E1 -11172.258,E2 -11172.258} C_VEL
LIN {X 0,Y 397.112,Z 154.018,A -85,B 0,C 180,E1 -11175.395,E2 -11175.395} C_VEL
LIN {X 0,Y 397.085,Z 154.019,A -85,B 0,C 180,E1 -11178.577,E2 -11178.577} C_VEL
LIN {X 0,Y 397.09,Z 154.023,A -85,B 0,C 180,E1 -11181.819,E2 -11181.819} C_VEL
LIN {X 0,Y 397.104,Z 154.018,A -85,B 0,C 180,E1 -11185.135,E2 -11185.135} C_VEL
LIN {X 0,Y 397.062,Z 154.021,A -85,B 0,C 180,E1 -11188.548,E2 -11188.548} C_VEL
LIN {X 0,Y 397.077,Z 154.022,A -85,B 0,C 180,E1 -11191.834,E2 -11191.834} C_VEL
LIN {X 0,Y 397.117,Z 154.015,A -85,B 0,C 180,E1 -11194.494,E2 -11194.494} C_VEL
LIN {X 0,Y 397.091,Z 154.018,A -85,B 0,C 180,E1 -11198.277,E2 -11198.277} C_VEL
LIN {X 0,Y 397.053,Z 154.023,A -85,B 0,C 180,E1 -11201.976,E2 -11201.976} C_VEL
LIN {X 0,Y 397.088,Z 154.025,A -85,B 0,C 180,E1 -11205.069,E2 -11205.069} C_VEL
LIN {X 0,Y 397.052,Z 154.023,A -85,B 0,C 180,E1 -11208.024,E2 -11208.024} C_VEL
LIN {X 0,Y 397.09,Z 154.018,A -85,B 0,C 180,E1 -11211.723,E2 -11211.723} C_VEL
LIN {X 0,Y 397.116,Z 154.015,A -85,B 0,C 180,E1 -11215.505,E2 -11215.505} C_VEL
LIN {X 0,Y 397.072,Z 154.025,A -85,B 0,C 180,E1 -11219.117,E2 -11219.117} C_VEL
LIN {X 0,Y 397.097,Z 154.155,A -85,B 0,C 180,E1 -11222.066,E2 -11222.066} C_VEL
LIN {X 0,Y 399.693,Z 166.873,A -85,B 0,C 180,E1 -11225.039,E2 -11225.039} C_VEL
LIN {X 0,Y 400.168,Z 171.987,A -85,B 0,C 180,E1 -11226.175,E2 -11226.175} C_VEL
LIN {X 0,Y 399.013,Z 188.456,A -85,B 0,C 180,E1 -11229.643,E2 -11229.643} C_VEL
LIN {X 0,Y 398.839,Z 190.841,A -85,B 0,C 180,E1 -11230.104,E2 -11230.104} C_VEL
LIN {X 0,Y 403.148,Z 219.393,A -85,B 0,C 180,E1 -11230.855,E2 -11230.855} C_VEL
LIN {X 0,Y 402.072,Z 299.25,A -85,B 0,C 180,E1 -11232.352,E2 -11232.352} C_VEL
LIN {X 0,Y 401.502,Z 313.019,A -85,B 0,C 180,E1 -11232.819,E2 -11232.819} C_VEL
LIN {X 0,Y 400.824,Z 325.437,A -85,B 0,C 180,E1 -11233.445,E2 -11233.445} C_VEL
LIN {X 0,Y 400.022,Z 336.542,A -85,B 0,C 180,E1 -11234.197,E2 -11234.197} C_VEL
LIN {X 0,Y 399.186,Z 348.139,A -85,B 0,C 180,E1 -11235.209,E2 -11235.209} C_VEL
LIN {X 0,Y 398.46,Z 358.328,A -85,B 0,C 180,E1 -11236.323,E2 -11236.323} C_VEL
LIN {X 0,Y 397.801,Z 367.137,A -85,B 0,C 180,E1 -11237.501,E2 -11237.501} C_VEL
LIN {X 0,Y 396.961,Z 376.376,A -85,B 0,C 180,E1 -11239.028,E2 -11239.028} C_VEL
LIN {X 0,Y 396.469,Z 383.81,A -85,B 0,C 180,E1 -11240.563,E2 -11240.563} C_VEL
LIN {X 0,Y 396.174,Z 388.854,A -85,B 0,C 180,E1 -11241.841,E2 -11241.841} C_VEL
LIN {X 0,Y 395.919,Z 393.742,A -85,B 0,C 180,E1 -11243.375,E2 -11243.375} C_VEL
LIN {X 0,Y 395.84,Z 397.489,A -85,B 0,C 180,E1 -11244.907,E2 -11244.907} C_VEL
LIN {X 0,Y 395.774,Z 399.419,A -85,B 0,C 180,E1 -11245.927,E2 -11245.927} C_VEL
LIN {X 0,Y 395.728,Z 400.912,A -85,B 0,C 180,E1 -11246.946,E2 -11246.946} C_VEL
LIN {X 0,Y 395.763,Z 401.956,A -85,B 0,C 180,E1 -11247.965,E2 -11247.965} C_VEL
LIN {X 0,Y 395.792,Z 402.606,A -85,B 0,C 180,E1 -11248.983,E2 -11248.983} C_VEL
LIN {X 0,Y 395.78,Z 402.863,A -85,B 0,C 180,E1 -11250,E2 -11250} C_VEL
LIN {X 0,Y 395.792,Z 402.713,A -85,B 0,C 180,E1 -11251.017,E2 -11251.017} C_VEL
LIN {X 0,Y 395.762,Z 402.129,A -85,B 0,C 180,E1 -11252.035,E2 -11252.035} C_VEL
LIN {X 0,Y 395.774,Z 399.783,A -85,B 0,C 180,E1 -11254.073,E2 -11254.073} C_VEL
LIN {X 0,Y 395.824,Z 396.458,A -85,B 0,C 180,E1 -11255.801,E2 -11255.801} C_VEL
LIN {X 0,Y 396.072,Z 391.391,A -85,B 0,C 180,E1 -11257.648,E2 -11257.648} C_VEL
LIN {X 0,Y 396.504,Z 384.889,A -85,B 0,C 180,E1 -11259.437,E2 -11259.437} C_VEL
LIN {X 0,Y 397.033,Z 377.782,A -85,B 0,C 180,E1 -11260.97,E2 -11260.97} C_VEL
LIN {X 0,Y 397.897,Z 368.914,A -85,B 0,C 180,E1 -11262.496,E2 -11262.496} C_VEL
LIN {X 0,Y 398.592,Z 360.129,A -85,B 0,C 180,E1 -11263.732,E2 -11263.732} C_VEL
LIN {X 0,Y 399.448,Z 350.22,A -85,B 0,C 180,E1 -11264.872,E2 -11264.872} C_VEL
LIN {X 0,Y 400.38,Z 338.784,A -85,B 0,C 180,E1 -11265.919,E2 -11265.919} C_VEL
LIN {X 0,Y 401.289,Z 326.406,A -85,B 0,C 180,E1 -11266.797,E2 -11266.797} C_VEL
LIN {X 0,Y 402.005,Z 314.688,A -85,B 0,C 180,E1 -11267.421,E2 -11267.421} C_VEL
LIN {X 0,Y 402.658,Z 302.107,A -85,B 0,C 180,E1 -11267.884,E2 -11267.884} C_VEL
LIN {X 0,Y 403.05,Z 284.725,A -85,B 0,C 180,E1 -11268.26,E2 -11268.26} C_VEL
LIN {X 0,Y 403.875,Z 218.007,A -85,B 0,C 180,E1 -11269.509,E2 -11269.509} C_VEL
LIN {X 0,Y 399.922,Z 194.118,A -85,B 0,C 180,E1 -11270.2,E2 -11270.2} C_VEL
LIN {X 0,Y 399.143,Z 189.76,A -85,B 0,C 180,E1 -11270.36,E2 -11270.36} C_VEL
LIN {X 0,Y 400.509,Z 171.683,A -85,B 0,C 180,E1 -11274.15,E2 -11274.15} C_VEL
LIN {X 0,Y 399.068,Z 163.116,A -85,B 0,C 180,E1 -11276.122,E2 -11276.122} C_VEL
LIN {X 0,Y 397.086,Z 154.026,A -85,B 0,C 180,E1 -11278.336,E2 -11278.336} C_VEL
LIN {X 0,Y 397.072,Z 154.028,A -85,B 0,C 180,E1 -11280.883,E2 -11280.883} C_VEL
LIN {X 0,Y 397.116,Z 154.021,A -85,B 0,C 180,E1 -11284.495,E2 -11284.495} C_VEL
LIN {X 0,Y 397.087,Z 154.021,A -85,B 0,C 180,E1 -11288.277,E2 -11288.277} C_VEL
LIN {X 0,Y 397.047,Z 154.031,A -85,B 0,C 180,E1 -11290.914,E2 -11290.914} C_VEL
LIN {X 0,Y 397.088,Z 154.022,A -85,B 0,C 180,E1 -11293.651,E2 -11293.651} C_VEL
LIN {X 0,Y 397.092,Z 154.023,A -85,B 0,C 180,E1 -11296.523,E2 -11296.523} C_VEL
LIN {X 0,Y 397.086,Z 154.018,A -85,B 0,C 180,E1 -11300.419,E2 -11300.419} C_VEL
LIN {X 0,Y 397.094,Z 154.018,A -85,B 0,C 180,E1 -11303.004,E2 -11303.004} C_VEL
LIN {X 0,Y 397.112,Z 154.015,A -85,B 0,C 180,E1 -11306.727,E2 -11306.727} C_VEL
LIN {X 0,Y 397.116,Z 154.016,A -85,B 0,C 180,E1 -11310.295,E2 -11310.295} C_VEL
LIN {X 0,Y 397.073,Z 154.02,A -85,B 0,C 180,E1 -11313.737,E2 -11313.737} C_VEL
LIN {X 0,Y 397.102,Z 154.019,A -85,B 0,C 180,E1 -11317.085,E2 -11317.085} C_VEL
LIN {X 0,Y 397.097,Z 154.014,A -85,B 0,C 180,E1 -11320.35,E2 -11320.35} C_VEL
LIN {X 0,Y 397.118,Z 154.012,A -85,B 0,C 180,E1 -11323.551,E2 -11323.551} C_VEL
LIN {X 0,Y 397.194,Z 154.008,A -85,B 0,C 180,E1 -11326.702,E2 -11326.702} C_VEL
LIN {X 0,Y 397.206,Z 153.999,A -85,B 0,C 180,E1 -11329.809,E2 -11329.809} C_VEL
LIN {X 0,Y 397.295,Z 153.986,A -85,B 0,C 180,E1 -11332.887,E2 -11332.887} C_VEL
LIN {X 0,Y 397.229,Z 154,A -85,B 0,C 180,E1 -11334.925,E2 -11334.925} C_VEL
LIN {X 0,Y 397.442,Z 153.971,A -85,B 0,C 180,E1 -11337.973,E2 -11337.973} C_VEL
LIN {X 0,Y 397.322,Z 153.987,A -85,B 0,C 180,E1 -11341.014,E2 -11341.014} C_VEL
LIN {X 0,Y 397.3,Z 153.992,A -85,B 0,C 180,E1 -11343.042,E2 -11343.042} C_VEL
LIN {X 0,Y 397.299,Z 153.991,A -85,B 0,C 180,E1 -11346.479,E2 -11346.479} C_VEL
LIN {X 0,Y 397.231,Z 153.999,A -85,B 0,C 180,E1 -11349.162,E2 -11349.162} C_VEL
LIN {X 0,Y 397.218,Z 154.003,A -85,B 0,C 180,E1 -11352.258,E2 -11352.258} C_VEL
LIN {X 0,Y 397.127,Z 154.017,A -85,B 0,C 180,E1 -11355.394,E2 -11355.394} C_VEL
LIN {X 0,Y 397.091,Z 154.02,A -85,B 0,C 180,E1 -11358.577,E2 -11358.577} C_VEL
LIN {X 0,Y 397.094,Z 154.023,A -85,B 0,C 180,E1 -11361.819,E2 -11361.819} C_VEL
LIN {X 0,Y 397.1,Z 154.023,A -85,B 0,C 180,E1 -11365.136,E2 -11365.136} C_VEL
LIN {X 0,Y 397.066,Z 154.026,A -85,B 0,C 180,E1 -11368.548,E2 -11368.548} C_VEL
LIN {X 0,Y 397.083,Z 154.025,A -85,B 0,C 180,E1 -11371.836,E2 -11371.836} C_VEL
LIN {X 0,Y 397.136,Z 154.054,A -85,B 0,C 180,E1 -11373.675,E2 -11373.675} C_VEL
LIN {X 0,Y 399.384,Z 165.052,A -85,B 0,C 180,E1 -11376.462,E2 -11376.462} C_VEL
LIN {X 0,Y 399.723,Z 169.113,A -85,B 0,C 180,E1 -11377.437,E2 -11377.437} C_VEL
LIN {X 0,Y 399.648,Z 170.455,A -85,B 0,C 180,E1 -11377.745,E2 -11377.745} C_VEL
LIN {X 0,Y 404.057,Z 191.212,A -85,B 0,C 180,E1 -11378.415,E2 -11378.415} C_VEL
LIN {X 0,Y 404.368,Z 195.312,A -85,B 0,C 180,E1 -11378.513,E2 -11378.513} C_VEL
LIN {X 0,Y 402.915,Z 278.539,A -85,B 0,C 180,E1 -11380.084,E2 -11380.084} C_VEL
LIN {X 0,Y 402.412,Z 292.27,A -85,B 0,C 180,E1 -11380.56,E2 -11380.56} C_VEL
LIN {X 0,Y 401.828,Z 305.104,A -85,B 0,C 180,E1 -11381.229,E2 -11381.229} C_VEL
LIN {X 0,Y 400.966,Z 317.245,A -85,B 0,C 180,E1 -11382.083,E2 -11382.083} C_VEL
LIN {X 0,Y 400.101,Z 328.887,A -85,B 0,C 180,E1 -11383.143,E2 -11383.143} C_VEL
LIN {X 0,Y 399.181,Z 339.498,A -85,B 0,C 180,E1 -11384.371,E2 -11384.371} C_VEL
LIN {X 0,Y 398.287,Z 349.481,A -85,B 0,C 180,E1 -11385.813,E2 -11385.813} C_VEL
LIN {X 0,Y 397.607,Z 356.788,A -85,B 0,C 180,E1 -11387.116,E2 -11387.116} C_VEL
LIN {X 0,Y 396.951,Z 364.359,A -85,B 0,C 180,E1 -11388.797,E2 -11388.797} C_VEL
LIN {X 0,Y 396.486,Z 369.87,A -85,B 0,C 180,E1 -11390.347,E2 -11390.347} C_VEL
LIN {X 0,Y 396.085,Z 375.028,A -85,B 0,C 180,E1 -11392.254,E2 -11392.254} C_VEL
LIN {X 0,Y 395.792,Z 378.473,A -85,B 0,C 180,E1 -11394.128,E2 -11394.128} C_VEL
LIN {X 0,Y 395.627,Z 379.983,A -85,B 0,C 180,E1 -11395.357,E2 -11395.357} C_VEL
LIN {X 0,Y 395.565,Z 380.882,A -85,B 0,C 180,E1 -11396.621,E2 -11396.621} C_VEL
LIN {X 0,Y 395.569,Z 381.11,A -85,B 0,C 180,E1 -11398.519,E2 -11398.519} C_VEL
LIN {X 0,Y 395.653,Z 379.861,A -85,B 0,C 180,E1 -11400.504,E2 -11400.504} C_VEL
LIN {X 0,Y 395.871,Z 377.006,A -85,B 0,C 180,E1 -11402.51,E2 -11402.51} C_VEL
LIN {X 0,Y 396.131,Z 373.217,A -85,B 0,C 180,E1 -11404.236,E2 -11404.236} C_VEL
LIN {X 0,Y 396.474,Z 368.093,A -85,B 0,C 180,E1 -11405.939,E2 -11405.939} C_VEL
LIN {X 0,Y 396.926,Z 361.452,A -85,B 0,C 180,E1 -11407.634,E2 -11407.634} C_VEL
LIN {X 0,Y 397.577,Z 353.183,A -85,B 0,C 180,E1 -11409.296,E2 -11409.296} C_VEL
LIN {X 0,Y 398.332,Z 344.492,A -85,B 0,C 180,E1 -11410.681,E2 -11410.681} C_VEL
LIN {X 0,Y 399.08,Z 334.437,A -85,B 0,C 180,E1 -11411.984,E2 -11411.984} C_VEL
LIN {X 0,Y 399.884,Z 324.618,A -85,B 0,C 180,E1 -11413.011,E2 -11413.011} C_VEL
LIN {X 0,Y 400.613,Z 313.693,A -85,B 0,C 180,E1 -11413.931,E2 -11413.931} C_VEL
LIN {X 0,Y 401.222,Z 301.794,A -85,B 0,C 180,E1 -11414.708,E2 -11414.708} C_VEL
LIN {X 0,Y 401.832,Z 288.865,A -85,B 0,C 180,E1 -11415.325,E2 -11415.325} C_VEL
LIN {X 0,Y 402.215,Z 276.782,A -85,B 0,C 180,E1 -11415.711,E2 -11415.711} C_VEL
LIN {X 0,Y 403.481,Z 192.568,A -85,B 0,C 180,E1 -11417.274,E2 -11417.274} C_VEL
LIN {X 0,Y 399.181,Z 170.103,A -85,B 0,C 180,E1 -11417.932,E2 -11417.932} C_VEL
LIN {X 0,Y 399.314,Z 165.205,A -85,B 0,C 180,E1 -11419.094,E2 -11419.094} C_VEL
LIN {X 0,Y 398.903,Z 162.979,A -85,B 0,C 180,E1 -11419.652,E2 -11419.652} C_VEL
LIN {X 0,Y 397.814,Z 161.373,A -85,B 0,C 180,E1 -11420.132,E2 -11420.132} C_VEL
LIN {X 0,Y 391.085,Z 156.729,A -85,B 0,C 180,E1 -11421.662,E2 -11421.662} C_VEL
LIN {X 0,Y 390.282,Z 154.868,A -85,B 0,C 180,E1 -11422.224,E2 -11422.224} C_VEL
LIN {X 0,Y 390.212,Z 154.878,A -85,B 0,C 180,E1 -11424.833,E2 -11424.833} C_VEL
LIN {X 0,Y 390.418,Z 154.851,A -85,B 0,C 180,E1 -11427.937,E2 -11427.937} C_VEL
LIN {X 0,Y 390.336,Z 154.86,A -85,B 0,C 180,E1 -11431.032,E2 -11431.032} C_VEL
LIN {X 0,Y 390.263,Z 154.869,A -85,B 0,C 180,E1 -11433.097,E2 -11433.097} C_VEL
LIN {X 0,Y 390.285,Z 154.872,A -85,B 0,C 180,E1 -11436.203,E2 -11436.203} C_VEL
LIN {X 0,Y 390.195,Z 154.877,A -85,B 0,C 180,E1 -11439.329,E2 -11439.329} C_VEL
LIN {X 0,Y 390.173,Z 154.882,A -85,B 0,C 180,E1 -11442.483,E2 -11442.483} C_VEL
LIN {X 0,Y 390.07,Z 154.896,A -85,B 0,C 180,E1 -11445.68,E2 -11445.68} C_VEL
LIN {X 0,Y 390.1,Z 154.889,A -85,B 0,C 180,E1 -11448.922,E2 -11448.922} C_VEL
LIN {X 0,Y 390.037,Z 154.899,A -85,B 0,C 180,E1 -11452.234,E2 -11452.234} C_VEL
LIN {X 0,Y 390.052,Z 154.901,A -85,B 0,C 180,E1 -11455.722,E2 -11455.722} C_VEL
LIN {X 0,Y 390.03,Z 154.899,A -85,B 0,C 180,E1 -11459.112,E2 -11459.112} C_VEL
LIN {X 0,Y 390.044,Z 154.896,A -85,B 0,C 180,E1 -11462.722,E2 -11462.722} C_VEL
LIN {X 0,Y 390.056,Z 154.897,A -85,B 0,C 180,E1 -11465.825,E2 -11465.825} C_VEL
LIN {X 0,Y 390.04,Z 154.901,A -85,B 0,C 180,E1 -11469.212,E2 -11469.212} C_VEL
LIN {X 0,Y 390.033,Z 154.897,A -85,B 0,C 180,E1 -11472.372,E2 -11472.372} C_VEL
LIN {X 0,Y 390.043,Z 154.902,A -85,B 0,C 180,E1 -11475.354,E2 -11475.354} C_VEL
LIN {X 0,Y 390.018,Z 154.899,A -85,B 0,C 180,E1 -11478.185,E2 -11478.185} C_VEL
LIN {X 0,Y 390.062,Z 154.897,A -85,B 0,C 180,E1 -11480.904,E2 -11480.904} C_VEL
LIN {X 0,Y 390.072,Z 154.896,A -85,B 0,C 180,E1 -11484.792,E2 -11484.792} C_VEL
LIN {X 0,Y 390.024,Z 154.9,A -85,B 0,C 180,E1 -11488.496,E2 -11488.496} C_VEL
LIN {X 0,Y 390.032,Z 154.897,A -85,B 0,C 180,E1 -11492.063,E2 -11492.063} C_VEL
LIN {X 0,Y 390.046,Z 154.896,A -85,B 0,C 180,E1 -11495.517,E2 -11495.517} C_VEL
LIN {X 0,Y 390.058,Z 154.899,A -85,B 0,C 180,E1 -11498.878,E2 -11498.878} C_VEL
LIN {X 0,Y 390.071,Z 154.894,A -85,B 0,C 180,E1 -11502.164,E2 -11502.164} C_VEL
LIN {X 0,Y 390.095,Z 154.89,A -85,B 0,C 180,E1 -11505.391,E2 -11505.391} C_VEL
LIN {X 0,Y 390.174,Z 154.879,A -85,B 0,C 180,E1 -11507.517,E2 -11507.517} C_VEL
LIN {X 0,Y 390.193,Z 154.881,A -85,B 0,C 180,E1 -11510.671,E2 -11510.671} C_VEL
LIN {X 0,Y 390.286,Z 154.867,A -85,B 0,C 180,E1 -11513.797,E2 -11513.797} C_VEL
LIN {X 0,Y 390.411,Z 154.853,A -85,B 0,C 180,E1 -11517.937,E2 -11517.937} C_VEL
LIN {X 0,Y 390.41,Z 154.856,A -85,B 0,C 180,E1 -11522.063,E2 -11522.063} C_VEL
LIN {X 0,Y 390.279,Z 154.871,A -85,B 0,C 180,E1 -11526.203,E2 -11526.203} C_VEL
LIN {X 0,Y 390.189,Z 154.879,A -85,B 0,C 180,E1 -11529.329,E2 -11529.329} C_VEL
LIN {X 0,Y 390.157,Z 154.883,A -85,B 0,C 180,E1 -11532.484,E2 -11532.484} C_VEL
LIN {X 0,Y 390.056,Z 154.899,A -85,B 0,C 180,E1 -11535.68,E2 -11535.68} C_VEL
LIN {X 0,Y 390.043,Z 154.896,A -85,B 0,C 180,E1 -11538.925,E2 -11538.925} C_VEL
LIN {X 0,Y 390.032,Z 154.898,A -85,B 0,C 180,E1 -11542.235,E2 -11542.235} C_VEL
LIN {X 0,Y 390.053,Z 154.9,A -85,B 0,C 180,E1 -11545.722,E2 -11545.722} C_VEL
LIN {X 0,Y 390.024,Z 154.901,A -85,B 0,C 180,E1 -11549.112,E2 -11549.112} C_VEL
LIN {X 0,Y 390.04,Z 154.897,A -85,B 0,C 180,E1 -11552.722,E2 -11552.722} C_VEL
LIN {X 0,Y 390.043,Z 154.897,A -85,B 0,C 180,E1 -11555.822,E2 -11555.822} C_VEL
LIN {X 0,Y 390.038,Z 154.903,A -85,B 0,C 180,E1 -11559.212,E2 -11559.212} C_VEL
LIN {X 0,Y 390.031,Z 154.898,A -85,B 0,C 180,E1 -11562.372,E2 -11562.372} C_VEL
LIN {X 0,Y 390.043,Z 154.9,A -85,B 0,C 180,E1 -11565.354,E2 -11565.354} C_VEL
LIN {X 0,Y 390.015,Z 154.899,A -85,B 0,C 180,E1 -11568.184,E2 -11568.184} C_VEL
LIN {X 0,Y 390.058,Z 154.9,A -85,B 0,C 180,E1 -11570.903,E2 -11570.903} C_VEL
LIN {X 0,Y 390.069,Z 154.899,A -85,B 0,C 180,E1 -11574.791,E2 -11574.791} C_VEL
LIN {X 0,Y 390.018,Z 154.903,A -85,B 0,C 180,E1 -11578.495,E2 -11578.495} C_VEL
LIN {X 0,Y 390.06,Z 155.051,A -85,B 0,C 180,E1 -11581.802,E2 -11581.802} C_VEL
LIN {X 0,Y 392.903,Z 169.108,A -85,B 0,C 180,E1 -11585.143,E2 -11585.143} C_VEL
LIN {X 0,Y 393.227,Z 172.94,A -85,B 0,C 180,E1 -11586.008,E2 -11586.008} C_VEL
LIN {X 0,Y 392.115,Z 188.14,A -85,B 0,C 180,E1 -11589.269,E2 -11589.269} C_VEL
LIN {X 0,Y 391.952,Z 190.531,A -85,B 0,C 180,E1 -11589.766,E2 -11589.766} C_VEL
LIN {X 0,Y 396.379,Z 220.166,A -85,B 0,C 180,E1 -11590.562,E2 -11590.562} C_VEL
LIN {X 0,Y 395.256,Z 299.198,A -85,B 0,C 180,E1 -11592.071,E2 -11592.071} C_VEL
LIN {X 0,Y 394.67,Z 312.916,A -85,B 0,C 180,E1 -11592.546,E2 -11592.546} C_VEL
LIN {X 0,Y 393.94,Z 325.816,A -85,B 0,C 180,E1 -11593.214,E2 -11593.214} C_VEL
LIN {X 0,Y 393.063,Z 337.588,A -85,B 0,C 180,E1 -11594.043,E2 -11594.043} C_VEL
LIN {X 0,Y 392.18,Z 348.959,A -85,B 0,C 180,E1 -11595.072,E2 -11595.072} C_VEL
LIN {X 0,Y 391.37,Z 359.774,A -85,B 0,C 180,E1 -11596.31,E2 -11596.31} C_VEL
LIN {X 0,Y 390.519,Z 370.073,A -85,B 0,C 180,E1 -11597.792,E2 -11597.792} C_VEL
LIN {X 0,Y 389.847,Z 377.403,A -85,B 0,C 180,E1 -11599.089,E2 -11599.089} C_VEL
LIN {X 0,Y 389.363,Z 384.616,A -85,B 0,C 180,E1 -11600.651,E2 -11600.651} C_VEL
LIN {X 0,Y 389.017,Z 390.354,A -85,B 0,C 180,E1 -11602.213,E2 -11602.213} C_VEL
LIN {X 0,Y 388.774,Z 395.066,A -85,B 0,C 180,E1 -11603.857,E2 -11603.857} C_VEL
LIN {X 0,Y 388.736,Z 397.241,A -85,B 0,C 180,E1 -11604.814,E2 -11604.814} C_VEL
LIN {X 0,Y 388.698,Z 399.181,A -85,B 0,C 180,E1 -11605.853,E2 -11605.853} C_VEL
LIN {X 0,Y 388.635,Z 400.689,A -85,B 0,C 180,E1 -11606.89,E2 -11606.89} C_VEL
LIN {X 0,Y 388.662,Z 401.742,A -85,B 0,C 180,E1 -11607.927,E2 -11607.927} C_VEL
LIN {X 0,Y 388.703,Z 402.4,A -85,B 0,C 180,E1 -11608.964,E2 -11608.964} C_VEL
LIN {X 0,Y 388.709,Z 402.665,A -85,B 0,C 180,E1 -11610,E2 -11610} C_VEL
LIN {X 0,Y 388.703,Z 402.527,A -85,B 0,C 180,E1 -11611.036,E2 -11611.036} C_VEL
LIN {X 0,Y 388.66,Z 401.952,A -85,B 0,C 180,E1 -11612.073,E2 -11612.073} C_VEL
LIN {X 0,Y 388.698,Z 399.618,A -85,B 0,C 180,E1 -11614.148,E2 -11614.148} C_VEL
LIN {X 0,Y 388.724,Z 396.644,A -85,B 0,C 180,E1 -11615.75,E2 -11615.75} C_VEL
LIN {X 0,Y 388.936,Z 392.818,A -85,B 0,C 180,E1 -11617.267,E2 -11617.267} C_VEL
LIN {X 0,Y 389.262,Z 387.767,A -85,B 0,C 180,E1 -11618.828,E2 -11618.828} C_VEL
LIN {X 0,Y 389.778,Z 381.431,A -85,B 0,C 180,E1 -11620.388,E2 -11620.388} C_VEL
LIN {X 0,Y 390.462,Z 373.505,A -85,B 0,C 180,E1 -11621.946,E2 -11621.946} C_VEL
LIN {X 0,Y 391.294,Z 365.435,A -85,B 0,C 180,E1 -11623.238,E2 -11623.238} C_VEL
LIN {X 0,Y 392.099,Z 355.603,A -85,B 0,C 180,E1 -11624.533,E2 -11624.533} C_VEL
LIN {X 0,Y 393.069,Z 344.67,A -85,B 0,C 180,E1 -11625.69,E2 -11625.69} C_VEL
LIN {X 0,Y 393.907,Z 333.99,A -85,B 0,C 180,E1 -11626.587,E2 -11626.587} C_VEL
LIN {X 0,Y 394.955,Z 321.171,A -85,B 0,C 180,E1 -11627.408,E2 -11627.408} C_VEL
LIN {X 0,Y 395.628,Z 308.26,A -85,B 0,C 180,E1 -11628.012,E2 -11628.012} C_VEL
LIN {X 0,Y 396.211,Z 295.614,A -85,B 0,C 180,E1 -11628.385,E2 -11628.385} C_VEL
LIN {X 0,Y 397.216,Z 218.51,A -85,B 0,C 180,E1 -11629.868,E2 -11629.868} C_VEL
LIN {X 0,Y 393.001,Z 193.36,A -85,B 0,C 180,E1 -11630.618,E2 -11630.618} C_VEL
LIN {X 0,Y 392.297,Z 189.536,A -85,B 0,C 180,E1 -11630.77,E2 -11630.77} C_VEL
LIN {X 0,Y 393.596,Z 173.253,A -85,B 0,C 180,E1 -11634.248,E2 -11634.248} C_VEL
LIN {X 0,Y 392.537,Z 166.276,A -85,B 0,C 180,E1 -11635.873,E2 -11635.873} C_VEL
LIN {X 0,Y 390.049,Z 154.902,A -85,B 0,C 180,E1 -11638.681,E2 -11638.681} C_VEL
LIN {X 0,Y 390.026,Z 154.906,A -85,B 0,C 180,E1 -11642.123,E2 -11642.123} C_VEL
LIN {X 0,Y 390.068,Z 154.899,A -85,B 0,C 180,E1 -11645.209,E2 -11645.209} C_VEL
LIN {X 0,Y 390.055,Z 154.902,A -85,B 0,C 180,E1 -11649.097,E2 -11649.097} C_VEL
LIN {X 0,Y 390.03,Z 154.9,A -85,B 0,C 180,E1 -11652.372,E2 -11652.372} C_VEL
LIN {X 0,Y 390.042,Z 154.903,A -85,B 0,C 180,E1 -11655.354,E2 -11655.354} C_VEL
LIN {X 0,Y 390.015,Z 154.901,A -85,B 0,C 180,E1 -11658.184,E2 -11658.184} C_VEL
LIN {X 0,Y 390.056,Z 154.897,A -85,B 0,C 180,E1 -11660.903,E2 -11660.903} C_VEL
LIN {X 0,Y 390.069,Z 154.897,A -85,B 0,C 180,E1 -11664.791,E2 -11664.791} C_VEL
LIN {X 0,Y 390.019,Z 154.901,A -85,B 0,C 180,E1 -11668.495,E2 -11668.495} C_VEL
LIN {X 0,Y 390.018,Z 154.897,A -85,B 0,C 180,E1 -11672.003,E2 -11672.003} C_VEL
LIN {X 0,Y 390.038,Z 154.892,A -85,B 0,C 180,E1 -11675.516,E2 -11675.516} C_VEL
LIN {X 0,Y 390.05,Z 154.89,A -85,B 0,C 180,E1 -11678.877,E2 -11678.877} C_VEL
LIN {X 0,Y 390.074,Z 154.893,A -85,B 0,C 180,E1 -11682.73,E2 -11682.73} C_VEL
LIN {X 0,Y 390.135,Z 154.889,A -85,B 0,C 180,E1 -11686.601,E2 -11686.601} C_VEL
LIN {X 0,Y 390.158,Z 154.876,A -85,B 0,C 180,E1 -11689.623,E2 -11689.623} C_VEL
LIN {X 0,Y 390.248,Z 154.865,A -85,B 0,C 180,E1 -11692.758,E2 -11692.758} C_VEL
LIN {X 0,Y 390.2,Z 154.876,A -85,B 0,C 180,E1 -11694.833,E2 -11694.833} C_VEL
LIN {X 0,Y 390.408,Z 154.846,A -85,B 0,C 180,E1 -11697.937,E2 -11697.937} C_VEL
LIN {X 0,Y 390.407,Z 154.849,A -85,B 0,C 180,E1 -11702.063,E2 -11702.063} C_VEL
LIN {X 0,Y 390.259,Z 154.868,A -85,B 0,C 180,E1 -11706.471,E2 -11706.471} C_VEL
LIN {X 0,Y 390.189,Z 154.877,A -85,B 0,C 180,E1 -11709.329,E2 -11709.329} C_VEL
LIN {X 0,Y 390.199,Z 154.877,A -85,B 0,C 180,E1 -11713.438,E2 -11713.438} C_VEL
LIN {X 0,Y 390.075,Z 154.896,A -85,B 0,C 180,E1 -11717.271,E2 -11717.271} C_VEL
LIN {X 0,Y 390.053,Z 154.897,A -85,B 0,C 180,E1 -11721.123,E2 -11721.123} C_VEL
LIN {X 0,Y 390.046,Z 154.9,A -85,B 0,C 180,E1 -11724.483,E2 -11724.483} C_VEL
LIN {X 0,Y 390.018,Z 154.907,A -85,B 0,C 180,E1 -11727.997,E2 -11727.997} C_VEL
LIN {X 0,Y 390.025,Z 154.905,A -85,B 0,C 180,E1 -11731.504,E2 -11731.504} C_VEL
LIN {X 0,Y 390.096,Z 154.923,A -85,B 0,C 180,E1 -11733.332,E2 -11733.332} C_VEL
LIN {X 0,Y 392.474,Z 166.468,A -85,B 0,C 180,E1 -11736.311,E2 -11736.311} C_VEL
LIN {X 0,Y 392.833,Z 170.683,A -85,B 0,C 180,E1 -11737.344,E2 -11737.344} C_VEL
LIN {X 0,Y 397.304,Z 191.435,A -85,B 0,C 180,E1 -11738.036,E2 -11738.036} C_VEL
LIN {X 0,Y 397.762,Z 194.82,A -85,B 0,C 180,E1 -11738.13,E2 -11738.13} C_VEL
LIN {X 0,Y 396.246,Z 278.372,A -85,B 0,C 180,E1 -11739.732,E2 -11739.732} C_VEL
LIN {X 0,Y 395.719,Z 292.059,A -85,B 0,C 180,E1 -11740.209,E2 -11740.209} C_VEL
LIN {X 0,Y 395.167,Z 304.036,A -85,B 0,C 180,E1 -11740.83,E2 -11740.83} C_VEL
LIN {X 0,Y 394.37,Z 315.681,A -85,B 0,C 180,E1 -11741.635,E2 -11741.635} C_VEL
LIN {X 0,Y 393.394,Z 327.483,A -85,B 0,C 180,E1 -11742.694,E2 -11742.694} C_VEL
LIN {X 0,Y 392.435,Z 337.97,A -85,B 0,C 180,E1 -11743.877,E2 -11743.877} C_VEL
LIN {X 0,Y 391.589,Z 347.441,A -85,B 0,C 180,E1 -11745.216,E2 -11745.216} C_VEL
LIN {X 0,Y 390.84,Z 355.15,A -85,B 0,C 180,E1 -11746.545,E2 -11746.545} C_VEL
LIN {X 0,Y 390.092,Z 362.899,A -85,B 0,C 180,E1 -11748.194,E2 -11748.194} C_VEL
LIN {X 0,Y 389.519,Z 368.976,A -85,B 0,C 180,E1 -11749.832,E2 -11749.832} C_VEL
LIN {X 0,Y 389.116,Z 373.781,A -85,B 0,C 180,E1 -11751.515,E2 -11751.515} C_VEL
LIN {X 0,Y 388.797,Z 377.645,A -85,B 0,C 180,E1 -11753.379,E2 -11753.379} C_VEL
LIN {X 0,Y 388.607,Z 379.488,A -85,B 0,C 180,E1 -11754.639,E2 -11754.639} C_VEL
LIN {X 0,Y 388.478,Z 380.968,A -85,B 0,C 180,E1 -11756.325,E2 -11756.325} C_VEL
LIN {X 0,Y 388.473,Z 381.33,A -85,B 0,C 180,E1 -11758.355,E2 -11758.355} C_VEL
LIN {X 0,Y 388.557,Z 380.317,A -85,B 0,C 180,E1 -11760.25,E2 -11760.25} C_VEL
LIN {X 0,Y 388.743,Z 377.561,A -85,B 0,C 180,E1 -11762.358,E2 -11762.358} C_VEL
LIN {X 0,Y 389.056,Z 373.447,A -85,B 0,C 180,E1 -11764.307,E2 -11764.307} C_VEL
LIN {X 0,Y 389.402,Z 368.34,A -85,B 0,C 180,E1 -11766.041,E2 -11766.041} C_VEL
LIN {X 0,Y 389.878,Z 361.751,A -85,B 0,C 180,E1 -11767.756,E2 -11767.756} C_VEL
LIN {X 0,Y 390.545,Z 354.018,A -85,B 0,C 180,E1 -11769.352,E2 -11769.352} C_VEL
LIN {X 0,Y 391.208,Z 346.65,A -85,B 0,C 180,E1 -11770.588,E2 -11770.588} C_VEL
LIN {X 0,Y 392.021,Z 336.463,A -85,B 0,C 180,E1 -11771.985,E2 -11771.985} C_VEL
LIN {X 0,Y 392.854,Z 326.335,A -85,B 0,C 180,E1 -11773.1,E2 -11773.1} C_VEL
LIN {X 0,Y 393.655,Z 315.228,A -85,B 0,C 180,E1 -11774.082,E2 -11774.082} C_VEL
LIN {X 0,Y 394.289,Z 303.526,A -85,B 0,C 180,E1 -11774.889,E2 -11774.889} C_VEL
LIN {X 0,Y 394.935,Z 290.57,A -85,B 0,C 180,E1 -11775.541,E2 -11775.541} C_VEL
LIN {X 0,Y 395.397,Z 277.422,A -85,B 0,C 180,E1 -11775.985,E2 -11775.985} C_VEL
LIN {X 0,Y 396.703,Z 193.299,A -85,B 0,C 180,E1 -11777.578,E2 -11777.578} C_VEL
LIN {X 0,Y 392.268,Z 170.264,A -85,B 0,C 180,E1 -11778.273,E2 -11778.273} C_VEL
LIN {X 0,Y 392.364,Z 166.592,A -85,B 0,C 180,E1 -11779.159,E2 -11779.159} C_VEL
LIN {X 0,Y 390.282,Z 154.868,A -85,B 0,C 180,E1 -11782.224,E2 -11782.224} C_VEL
LIN {X 0,Y 389.53,Z 154.965,A -85,B 0,C 180,E1 -11783.084,E2 -11783.084} C_VEL
LIN {X 0,Y 386.568,Z 155.335,A -85,B 0,C 180,E1 -11784.482,E2 -11784.482} C_VEL
LIN {X 0,Y 384.17,Z 155.629,A -85,B 0,C 180,E1 -11785.612,E2 -11785.612} C_VEL
LIN {X 0,Y 383.245,Z 155.749,A -85,B 0,C 180,E1 -11786.486,E2 -11786.486} C_VEL
LIN {X 0,Y 383.223,Z 155.747,A -85,B 0,C 180,E1 -11786.782,E2 -11786.782} C_VEL
LIN {X 0,Y 383.385,Z 155.727,A -85,B 0,C 180,E1 -11787.899,E2 -11787.899} C_VEL
LIN {X 0,Y 383.303,Z 155.736,A -85,B 0,C 180,E1 -11791.051,E2 -11791.051} C_VEL
LIN {X 0,Y 383.201,Z 155.748,A -85,B 0,C 180,E1 -11793.154,E2 -11793.154} C_VEL
LIN {X 0,Y 383.242,Z 155.749,A -85,B 0,C 180,E1 -11796.317,E2 -11796.317} C_VEL
LIN {X 0,Y 383.145,Z 155.756,A -85,B 0,C 180,E1 -11799.502,E2 -11799.502} C_VEL
LIN {X 0,Y 383.128,Z 155.759,A -85,B 0,C 180,E1 -11803.536,E2 -11803.536} C_VEL
LIN {X 0,Y 383.06,Z 155.767,A -85,B 0,C 180,E1 -11807.437,E2 -11807.437} C_VEL
LIN {X 0,Y 383.031,Z 155.77,A -85,B 0,C 180,E1 -11810.647,E2 -11810.647} C_VEL
LIN {X 0,Y 383.012,Z 155.778,A -85,B 0,C 180,E1 -11813.809,E2 -11813.809} C_VEL
LIN {X 0,Y 382.984,Z 155.778,A -85,B 0,C 180,E1 -11817.308,E2 -11817.308} C_VEL
LIN {X 0,Y 382.984,Z 155.776,A -85,B 0,C 180,E1 -11820.919,E2 -11820.919} C_VEL
LIN {X 0,Y 383.019,Z 155.771,A -85,B 0,C 180,E1 -11824.668,E2 -11824.668} C_VEL
LIN {X 0,Y 382.996,Z 155.776,A -85,B 0,C 180,E1 -11827.903,E2 -11827.903} C_VEL
LIN {X 0,Y 382.963,Z 155.784,A -85,B 0,C 180,E1 -11831.351,E2 -11831.351} C_VEL
LIN {X 0,Y 382.996,Z 155.774,A -85,B 0,C 180,E1 -11834.303,E2 -11834.303} C_VEL
LIN {X 0,Y 383.013,Z 155.778,A -85,B 0,C 180,E1 -11837.24,E2 -11837.24} C_VEL
LIN {X 0,Y 382.989,Z 155.775,A -85,B 0,C 180,E1 -11840.419,E2 -11840.419} C_VEL
LIN {X 0,Y 383.018,Z 155.771,A -85,B 0,C 180,E1 -11844.043,E2 -11844.043} C_VEL
LIN {X 0,Y 382.988,Z 155.776,A -85,B 0,C 180,E1 -11847.579,E2 -11847.579} C_VEL
LIN {X 0,Y 382.98,Z 155.777,A -85,B 0,C 180,E1 -11850.299,E2 -11850.299} C_VEL
LIN {X 0,Y 383.007,Z 155.773,A -85,B 0,C 180,E1 -11854.045,E2 -11854.045} C_VEL
LIN {X 0,Y 382.991,Z 155.775,A -85,B 0,C 180,E1 -11857.334,E2 -11857.334} C_VEL
LIN {X 0,Y 383.045,Z 155.774,A -85,B 0,C 180,E1 -11860.715,E2 -11860.715} C_VEL
LIN {X 0,Y 383.023,Z 155.772,A -85,B 0,C 180,E1 -11864.024,E2 -11864.024} C_VEL
LIN {X 0,Y 383.14,Z 155.756,A -85,B 0,C 180,E1 -11867.284,E2 -11867.284} C_VEL
LIN {X 0,Y 383.144,Z 155.761,A -85,B 0,C 180,E1 -11870.498,E2 -11870.498} C_VEL
LIN {X 0,Y 383.242,Z 155.744,A -85,B 0,C 180,E1 -11873.683,E2 -11873.683} C_VEL
LIN {X 0,Y 383.377,Z 155.729,A -85,B 0,C 180,E1 -11877.899,E2 -11877.899} C_VEL
LIN {X 0,Y 383.376,Z 155.733,A -85,B 0,C 180,E1 -11882.101,E2 -11882.101} C_VEL
LIN {X 0,Y 383.237,Z 155.747,A -85,B 0,C 180,E1 -11886.317,E2 -11886.317} C_VEL
LIN {X 0,Y 383.177,Z 155.753,A -85,B 0,C 180,E1 -11888.438,E2 -11888.438} C_VEL
LIN {X 0,Y 383.087,Z 155.766,A -85,B 0,C 180,E1 -11891.642,E2 -11891.642} C_VEL
LIN {X 0,Y 383.056,Z 155.772,A -85,B 0,C 180,E1 -11893.799,E2 -11893.799} C_VEL
LIN {X 0,Y 383.025,Z 155.773,A -85,B 0,C 180,E1 -11897.42,E2 -11897.42} C_VEL
LIN {X 0,Y 383.015,Z 155.771,A -85,B 0,C 180,E1 -11900.64,E2 -11900.64} C_VEL
LIN {X 0,Y 383.009,Z 155.776,A -85,B 0,C 180,E1 -11903.809,E2 -11903.809} C_VEL
LIN {X 0,Y 382.968,Z 155.781,A -85,B 0,C 180,E1 -11907.309,E2 -11907.309} C_VEL
LIN {X 0,Y 382.98,Z 155.777,A -85,B 0,C 180,E1 -11910.919,E2 -11910.919} C_VEL
LIN {X 0,Y 383.013,Z 155.772,A -85,B 0,C 180,E1 -11914.669,E2 -11914.669} C_VEL
LIN {X 0,Y 382.993,Z 155.775,A -85,B 0,C 180,E1 -11917.902,E2 -11917.902} C_VEL
LIN {X 0,Y 382.962,Z 155.783,A -85,B 0,C 180,E1 -11921.35,E2 -11921.35} C_VEL
LIN {X 0,Y 382.991,Z 155.775,A -85,B 0,C 180,E1 -11924.302,E2 -11924.302} C_VEL
LIN {X 0,Y 382.983,Z 155.78,A -85,B 0,C 180,E1 -11927.236,E2 -11927.236} C_VEL
LIN {X 0,Y 382.986,Z 155.776,A -85,B 0,C 180,E1 -11930.419,E2 -11930.419} C_VEL
LIN {X 0,Y 383.013,Z 155.772,A -85,B 0,C 180,E1 -11934.043,E2 -11934.043} C_VEL
LIN {X 0,Y 382.982,Z 155.776,A -85,B 0,C 180,E1 -11937.579,E2 -11937.579} C_VEL
LIN {X 0,Y 382.993,Z 155.78,A -85,B 0,C 180,E1 -11940.903,E2 -11940.903} C_VEL
LIN {X 0,Y 382.991,Z 155.846,A -85,B 0,C 180,E1 -11941.503,E2 -11941.503} C_VEL
LIN {X 0,Y 385.885,Z 170.039,A -85,B 0,C 180,E1 -11944.948,E2 -11944.948} C_VEL
LIN {X 0,Y 386.266,Z 174.179,A -85,B 0,C 180,E1 -11945.901,E2 -11945.901} C_VEL
LIN {X 0,Y 385.079,Z 189.715,A -85,B 0,C 180,E1 -11949.291,E2 -11949.291} C_VEL
LIN {X 0,Y 385.021,Z 190.256,A -85,B 0,C 180,E1 -11949.408,E2 -11949.408} C_VEL
LIN {X 0,Y 389.641,Z 220.446,A -85,B 0,C 180,E1 -11950.249,E2 -11950.249} C_VEL
LIN {X 0,Y 388.441,Z 299.144,A -85,B 0,C 180,E1 -11951.78,E2 -11951.78} C_VEL
LIN {X 0,Y 387.858,Z 312.815,A -85,B 0,C 180,E1 -11952.263,E2 -11952.263} C_VEL
LIN {X 0,Y 387.122,Z 325.175,A -85,B 0,C 180,E1 -11952.91,E2 -11952.91} C_VEL
LIN {X 0,Y 386.21,Z 337.045,A -85,B 0,C 180,E1 -11953.753,E2 -11953.753} C_VEL
LIN {X 0,Y 385.289,Z 348.48,A -85,B 0,C 180,E1 -11954.799,E2 -11954.799} C_VEL
LIN {X 0,Y 384.543,Z 358.362,A -85,B 0,C 180,E1 -11955.929,E2 -11955.929} C_VEL
LIN {X 0,Y 383.722,Z 368.062,A -85,B 0,C 180,E1 -11957.304,E2 -11957.304} C_VEL
LIN {X 0,Y 382.848,Z 377.063,A -85,B 0,C 180,E1 -11958.887,E2 -11958.887} C_VEL
LIN {X 0,Y 382.323,Z 384.308,A -85,B 0,C 180,E1 -11960.477,E2 -11960.477} C_VEL
LIN {X 0,Y 381.941,Z 390.075,A -85,B 0,C 180,E1 -11962.068,E2 -11962.068} C_VEL
LIN {X 0,Y 381.686,Z 395.142,A -85,B 0,C 180,E1 -11963.884,E2 -11963.884} C_VEL
LIN {X 0,Y 381.623,Z 398.943,A -85,B 0,C 180,E1 -11965.776,E2 -11965.776} C_VEL
LIN {X 0,Y 381.547,Z 400.464,A -85,B 0,C 180,E1 -11966.832,E2 -11966.832} C_VEL
LIN {X 0,Y 381.56,Z 401.528,A -85,B 0,C 180,E1 -11967.889,E2 -11967.889} C_VEL
LIN {X 0,Y 381.618,Z 402.193,A -85,B 0,C 180,E1 -11968.945,E2 -11968.945} C_VEL
LIN {X 0,Y 381.64,Z 402.467,A -85,B 0,C 180,E1 -11970,E2 -11970} C_VEL
LIN {X 0,Y 381.603,Z 402.34,A -85,B 0,C 180,E1 -11971.055,E2 -11971.055} C_VEL
LIN {X 0,Y 381.558,Z 401.774,A -85,B 0,C 180,E1 -11972.111,E2 -11972.111} C_VEL
LIN {X 0,Y 381.623,Z 399.453,A -85,B 0,C 180,E1 -11974.225,E2 -11974.225} C_VEL
LIN {X 0,Y 381.669,Z 395.993,A -85,B 0,C 180,E1 -11976.092,E2 -11976.092} C_VEL
LIN {X 0,Y 381.952,Z 391.129,A -85,B 0,C 180,E1 -11977.932,E2 -11977.932} C_VEL
LIN {X 0,Y 382.462,Z 384.656,A -85,B 0,C 180,E1 -11979.786,E2 -11979.786} C_VEL
LIN {X 0,Y 383.049,Z 377.606,A -85,B 0,C 180,E1 -11981.375,E2 -11981.375} C_VEL
LIN {X 0,Y 384.008,Z 368.793,A -85,B 0,C 180,E1 -11982.956,E2 -11982.956} C_VEL
LIN {X 0,Y 384.927,Z 358.557,A -85,B 0,C 180,E1 -11984.438,E2 -11984.438} C_VEL
LIN {X 0,Y 385.994,Z 347.351,A -85,B 0,C 180,E1 -11985.714,E2 -11985.714} C_VEL
LIN {X 0,Y 387.017,Z 335.812,A -85,B 0,C 180,E1 -11986.755,E2 -11986.755} C_VEL
LIN {X 0,Y 388.054,Z 323.684,A -85,B 0,C 180,E1 -11987.591,E2 -11987.591} C_VEL
LIN {X 0,Y 388.801,Z 310.268,A -85,B 0,C 180,E1 -11988.271,E2 -11988.271} C_VEL
LIN {X 0,Y 389.481,Z 297.94,A -85,B 0,C 180,E1 -11988.681,E2 -11988.681} C_VEL
LIN {X 0,Y 390.628,Z 219.552,A -85,B 0,C 180,E1 -11990.224,E2 -11990.224} C_VEL
LIN {X 0,Y 386.561,Z 195.13,A -85,B 0,C 180,E1 -11990.972,E2 -11990.972} C_VEL
LIN {X 0,Y 385.448,Z 189.325,A -85,B 0,C 180,E1 -11991.195,E2 -11991.195} C_VEL
LIN {X 0,Y 386.697,Z 174.322,A -85,B 0,C 180,E1 -11994.463,E2 -11994.463} C_VEL
LIN {X 0,Y 385.102,Z 165.478,A -85,B 0,C 180,E1 -11996.589,E2 -11996.589} C_VEL
LIN {X 0,Y 382.998,Z 155.781,A -85,B 0,C 180,E1 -11999.059,E2 -11999.059} C_VEL
LIN {X 0,Y 382.983,Z 155.784,A -85,B 0,C 180,E1 -12002.421,E2 -12002.421} C_VEL
LIN {X 0,Y 383.013,Z 155.774,A -85,B 0,C 180,E1 -12005.957,E2 -12005.957} C_VEL
LIN {X 0,Y 382.985,Z 155.779,A -85,B 0,C 180,E1 -12009.581,E2 -12009.581} C_VEL
LIN {X 0,Y 383.008,Z 155.778,A -85,B 0,C 180,E1 -12012.779,E2 -12012.779} C_VEL
LIN {X 0,Y 382.991,Z 155.778,A -85,B 0,C 180,E1 -12015.788,E2 -12015.788} C_VEL
LIN {X 0,Y 382.963,Z 155.785,A -85,B 0,C 180,E1 -12018.801,E2 -12018.801} C_VEL
LIN {X 0,Y 382.992,Z 155.776,A -85,B 0,C 180,E1 -12022.099,E2 -12022.099} C_VEL
LIN {X 0,Y 383.013,Z 155.774,A -85,B 0,C 180,E1 -12025.331,E2 -12025.331} C_VEL
LIN {X 0,Y 382.98,Z 155.778,A -85,B 0,C 180,E1 -12029.081,E2 -12029.081} C_VEL
LIN {X 0,Y 382.968,Z 155.782,A -85,B 0,C 180,E1 -12032.691,E2 -12032.691} C_VEL
LIN {X 0,Y 383.007,Z 155.77,A -85,B 0,C 180,E1 -12036.191,E2 -12036.191} C_VEL
LIN {X 0,Y 383.038,Z 155.76,A -85,B 0,C 180,E1 -12039.597,E2 -12039.597} C_VEL
LIN {X 0,Y 383.042,Z 155.767,A -85,B 0,C 180,E1 -12042.928,E2 -12042.928} C_VEL
LIN {X 0,Y 383.093,Z 155.767,A -85,B 0,C 180,E1 -12046.487,E2 -12046.487} C_VEL
LIN {X 0,Y 383.122,Z 155.751,A -85,B 0,C 180,E1 -12049.43,E2 -12049.43} C_VEL
LIN {X 0,Y 383.206,Z 155.743,A -85,B 0,C 180,E1 -12052.624,E2 -12052.624} C_VEL
LIN {X 0,Y 383.172,Z 155.753,A -85,B 0,C 180,E1 -12054.738,E2 -12054.738} C_VEL
LIN {X 0,Y 383.372,Z 155.722,A -85,B 0,C 180,E1 -12057.899,E2 -12057.899} C_VEL
LIN {X 0,Y 383.372,Z 155.725,A -85,B 0,C 180,E1 -12062.101,E2 -12062.101} C_VEL
LIN {X 0,Y 383.225,Z 155.745,A -85,B 0,C 180,E1 -12066.459,E2 -12066.459} C_VEL
LIN {X 0,Y 383.14,Z 155.755,A -85,B 0,C 180,E1 -12069.502,E2 -12069.502} C_VEL
LIN {X 0,Y 383.13,Z 155.759,A -85,B 0,C 180,E1 -12073.536,E2 -12073.536} C_VEL
LIN {X 0,Y 383.027,Z 155.775,A -85,B 0,C 180,E1 -12077.42,E2 -12077.42} C_VEL
LIN {X 0,Y 383.017,Z 155.772,A -85,B 0,C 180,E1 -12080.641,E2 -12080.641} C_VEL
LIN {X 0,Y 383.014,Z 155.778,A -85,B 0,C 180,E1 -12083.809,E2 -12083.809} C_VEL
LIN {X 0,Y 382.973,Z 155.785,A -85,B 0,C 180,E1 -12087.309,E2 -12087.309} C_VEL
LIN {X 0,Y 382.984,Z 155.781,A -85,B 0,C 180,E1 -12090.919,E2 -12090.919} C_VEL
LIN {X 0,Y 383.026,Z 155.869,A -85,B 0,C 180,E1 -12092.991,E2 -12092.991} C_VEL
LIN {X 0,Y 385.221,Z 166.197,A -85,B 0,C 180,E1 -12095.719,E2 -12095.719} C_VEL
LIN {X 0,Y 386,Z 171.114,A -85,B 0,C 180,E1 -12096.93,E2 -12096.93} C_VEL
LIN {X 0,Y 390.585,Z 191.711,A -85,B 0,C 180,E1 -12097.645,E2 -12097.645} C_VEL
LIN {X 0,Y 391.172,Z 195.821,A -85,B 0,C 180,E1 -12097.764,E2 -12097.764} C_VEL
LIN {X 0,Y 389.591,Z 278.8,A -85,B 0,C 180,E1 -12099.386,E2 -12099.386} C_VEL
LIN {X 0,Y 389.032,Z 292.384,A -85,B 0,C 180,E1 -12099.87,E2 -12099.87} C_VEL
LIN {X 0,Y 388.407,Z 304.957,A -85,B 0,C 180,E1 -12100.538,E2 -12100.538} C_VEL
LIN {X 0,Y 387.534,Z 316.691,A -85,B 0,C 180,E1 -12101.379,E2 -12101.379} C_VEL
LIN {X 0,Y 386.552,Z 328.327,A -85,B 0,C 180,E1 -12102.455,E2 -12102.455} C_VEL
LIN {X 0,Y 385.601,Z 338.195,A -85,B 0,C 180,E1 -12103.595,E2 -12103.595} C_VEL
LIN {X 0,Y 384.754,Z 346.95,A -85,B 0,C 180,E1 -12104.841,E2 -12104.841} C_VEL
LIN {X 0,Y 383.93,Z 355.167,A -85,B 0,C 180,E1 -12106.272,E2 -12106.272} C_VEL
LIN {X 0,Y 383.111,Z 363.003,A -85,B 0,C 180,E1 -12107.965,E2 -12107.965} C_VEL
LIN {X 0,Y 382.564,Z 368.297,A -85,B 0,C 180,E1 -12109.395,E2 -12109.395} C_VEL
LIN {X 0,Y 382.099,Z 373.789,A -85,B 0,C 180,E1 -12111.29,E2 -12111.29} C_VEL
LIN {X 0,Y 381.736,Z 377.807,A -85,B 0,C 180,E1 -12113.248,E2 -12113.248} C_VEL
LIN {X 0,Y 381.446,Z 380.334,A -85,B 0,C 180,E1 -12115.168,E2 -12115.168} C_VEL
LIN {X 0,Y 381.385,Z 381.239,A -85,B 0,C 180,E1 -12116.438,E2 -12116.438} C_VEL
LIN {X 0,Y 381.35,Z 381.588,A -85,B 0,C 180,E1 -12117.968,E2 -12117.968} C_VEL
LIN {X 0,Y 381.431,Z 380.721,A -85,B 0,C 180,E1 -12119.997,E2 -12119.997} C_VEL
LIN {X 0,Y 381.618,Z 378.241,A -85,B 0,C 180,E1 -12122.127,E2 -12122.127} C_VEL
LIN {X 0,Y 381.91,Z 375.072,A -85,B 0,C 180,E1 -12123.79,E2 -12123.79} C_VEL
LIN {X 0,Y 382.236,Z 370.41,A -85,B 0,C 180,E1 -12125.562,E2 -12125.562} C_VEL
LIN {X 0,Y 382.697,Z 364.358,A -85,B 0,C 180,E1 -12127.316,E2 -12127.316} C_VEL
LIN {X 0,Y 383.255,Z 357.481,A -85,B 0,C 180,E1 -12128.892,E2 -12128.892} C_VEL
LIN {X 0,Y 383.913,Z 350.444,A -85,B 0,C 180,E1 -12130.204,E2 -12130.204} C_VEL
LIN {X 0,Y 384.732,Z 341.35,A -85,B 0,C 180,E1 -12131.596,E2 -12131.596} C_VEL
LIN {X 0,Y 385.62,Z 330.678,A -85,B 0,C 180,E1 -12132.909,E2 -12132.909} C_VEL
LIN {X 0,Y 386.534,Z 319.135,A -85,B 0,C 180,E1 -12134.038,E2 -12134.038} C_VEL
LIN {X 0,Y 387.299,Z 307.612,A -85,B 0,C 180,E1 -12134.912,E2 -12134.912} C_VEL
LIN {X 0,Y 387.899,Z 294.948,A -85,B 0,C 180,E1 -12135.641,E2 -12135.641} C_VEL
LIN {X 0,Y 388.447,Z 282.786,A -85,B 0,C 180,E1 -12136.129,E2 -12136.129} C_VEL
LIN {X 0,Y 388.787,Z 268.057,A -85,B 0,C 180,E1 -12136.482,E2 -12136.482} C_VEL
LIN {X 0,Y 389.933,Z 194.137,A -85,B 0,C 180,E1 -12137.891,E2 -12137.891} C_VEL
LIN {X 0,Y 385.386,Z 170.411,A -85,B 0,C 180,E1 -12138.628,E2 -12138.628} C_VEL
LIN {X 0,Y 385.253,Z 166.961,A -85,B 0,C 180,E1 -12139.489,E2 -12139.489} C_VEL
LIN {X 0,Y 383.214,Z 155.748,A -85,B 0,C 180,E1 -12142.476,E2 -12142.476} C_VEL
LIN {X 0,Y 383.183,Z 155.755,A -85,B 0,C 180,E1 -12144.738,E2 -12144.738} C_VEL
LIN {X 0,Y 383.223,Z 155.747,A -85,B 0,C 180,E1 -12146.782,E2 -12146.782} C_VEL
LIN {X 0,Y 383.014,Z 155.777,A -85,B 0,C 180,E1 -12147.369,E2 -12147.369} C_VEL
LIN {X 0,Y 381.739,Z 155.938,A -85,B 0,C 180,E1 -12148.235,E2 -12148.235} C_VEL
LIN {X 0,Y 377.396,Z 156.476,A -85,B 0,C 180,E1 -12150.24,E2 -12150.24} C_VEL
LIN {X 0,Y 376.351,Z 156.602,A -85,B 0,C 180,E1 -12151.133,E2 -12151.133} C_VEL
LIN {X 0,Y 376.279,Z 156.61,A -85,B 0,C 180,E1 -12151.435,E2 -12151.435} C_VEL
LIN {X 0,Y 376.14,Z 156.628,A -85,B 0,C 180,E1 -12153.213,E2 -12153.213} C_VEL
LIN {X 0,Y 376.2,Z 156.624,A -85,B 0,C 180,E1 -12156.436,E2 -12156.436} C_VEL
LIN {X 0,Y 376.115,Z 156.633,A -85,B 0,C 180,E1 -12159.682,E2 -12159.682} C_VEL
LIN {X 0,Y 376.092,Z 156.636,A -85,B 0,C 180,E1 -12163.658,E2 -12163.658} C_VEL
LIN {X 0,Y 376.014,Z 156.646,A -85,B 0,C 180,E1 -12167.592,E2 -12167.592} C_VEL
LIN {X 0,Y 375.981,Z 156.648,A -85,B 0,C 180,E1 -12170.832,E2 -12170.832} C_VEL
LIN {X 0,Y 375.938,Z 156.655,A -85,B 0,C 180,E1 -12174.286,E2 -12174.286} C_VEL
LIN {X 0,Y 375.922,Z 156.655,A -85,B 0,C 180,E1 -12176.66,E2 -12176.66} C_VEL
LIN {X 0,Y 375.918,Z 156.656,A -85,B 0,C 180,E1 -12179.084,E2 -12179.084} C_VEL
LIN {X 0,Y 375.959,Z 156.656,A -85,B 0,C 180,E1 -12181.562,E2 -12181.562} C_VEL
LIN {X 0,Y 375.958,Z 156.656,A -85,B 0,C 180,E1 -12185.416,E2 -12185.416} C_VEL
LIN {X 0,Y 375.938,Z 156.653,A -85,B 0,C 180,E1 -12188.263,E2 -12188.263} C_VEL
LIN {X 0,Y 375.919,Z 156.659,A -85,B 0,C 180,E1 -12191.598,E2 -12191.598} C_VEL
LIN {X 0,Y 375.926,Z 156.656,A -85,B 0,C 180,E1 -12194.731,E2 -12194.731} C_VEL
LIN {X 0,Y 375.928,Z 156.656,A -85,B 0,C 180,E1 -12197.699,E2 -12197.699} C_VEL
LIN {X 0,Y 375.938,Z 156.654,A -85,B 0,C 180,E1 -12200.534,E2 -12200.534} C_VEL
LIN {X 0,Y 375.961,Z 156.652,A -85,B 0,C 180,E1 -12203.497,E2 -12203.497} C_VEL
LIN {X 0,Y 375.96,Z 156.65,A -85,B 0,C 180,E1 -12205.888,E2 -12205.888} C_VEL
LIN {X 0,Y 375.964,Z 156.65,A -85,B 0,C 180,E1 -12209.687,E2 -12209.687} C_VEL
LIN {X 0,Y 375.931,Z 156.654,A -85,B 0,C 180,E1 -12212.136,E2 -12212.136} C_VEL
LIN {X 0,Y 375.971,Z 156.649,A -85,B 0,C 180,E1 -12215.717,E2 -12215.717} C_VEL
LIN {X 0,Y 375.983,Z 156.649,A -85,B 0,C 180,E1 -12219.197,E2 -12219.197} C_VEL
LIN {X 0,Y 376.013,Z 156.65,A -85,B 0,C 180,E1 -12222.599,E2 -12222.599} C_VEL
LIN {X 0,Y 376.094,Z 156.638,A -85,B 0,C 180,E1 -12226.342,E2 -12226.342} C_VEL
LIN {X 0,Y 376.114,Z 156.636,A -85,B 0,C 180,E1 -12230.318,E2 -12230.318} C_VEL
LIN {X 0,Y 376.201,Z 156.62,A -85,B 0,C 180,E1 -12233.564,E2 -12233.564} C_VEL
LIN {X 0,Y 376.341,Z 156.605,A -85,B 0,C 180,E1 -12237.86,E2 -12237.86} C_VEL
LIN {X 0,Y 376.341,Z 156.61,A -85,B 0,C 180,E1 -12242.14,E2 -12242.14} C_VEL
LIN {X 0,Y 376.197,Z 156.623,A -85,B 0,C 180,E1 -12246.436,E2 -12246.436} C_VEL
LIN {X 0,Y 376.11,Z 156.635,A -85,B 0,C 180,E1 -12249.682,E2 -12249.682} C_VEL
LIN {X 0,Y 376.043,Z 156.644,A -85,B 0,C 180,E1 -12253.626,E2 -12253.626} C_VEL
LIN {X 0,Y 375.984,Z 156.652,A -85,B 0,C 180,E1 -12257.576,E2 -12257.576} C_VEL
LIN {X 0,Y 375.982,Z 156.648,A -85,B 0,C 180,E1 -12260.832,E2 -12260.832} C_VEL
LIN {X 0,Y 375.936,Z 156.654,A -85,B 0,C 180,E1 -12264.285,E2 -12264.285} C_VEL
LIN {X 0,Y 375.911,Z 156.656,A -85,B 0,C 180,E1 -12266.66,E2 -12266.66} C_VEL
LIN {X 0,Y 375.914,Z 156.658,A -85,B 0,C 180,E1 -12269.084,E2 -12269.084} C_VEL
LIN {X 0,Y 375.955,Z 156.656,A -85,B 0,C 180,E1 -12271.562,E2 -12271.562} C_VEL
LIN {X 0,Y 375.95,Z 156.657,A -85,B 0,C 180,E1 -12275.416,E2 -12275.416} C_VEL
LIN {X 0,Y 375.935,Z 156.653,A -85,B 0,C 180,E1 -12278.262,E2 -12278.262} C_VEL
LIN {X 0,Y 375.915,Z 156.658,A -85,B 0,C 180,E1 -12281.597,E2 -12281.597} C_VEL
LIN {X 0,Y 375.922,Z 156.658,A -85,B 0,C 180,E1 -12284.73,E2 -12284.73} C_VEL
LIN {X 0,Y 375.908,Z 156.657,A -85,B 0,C 180,E1 -12287.696,E2 -12287.696} C_VEL
LIN {X 0,Y 375.935,Z 156.656,A -85,B 0,C 180,E1 -12290.534,E2 -12290.534} C_VEL
LIN {X 0,Y 375.958,Z 156.651,A -85,B 0,C 180,E1 -12293.497,E2 -12293.497} C_VEL
LIN {X 0,Y 375.958,Z 156.65,A -85,B 0,C 180,E1 -12295.888,E2 -12295.888} C_VEL
LIN {X 0,Y 375.96,Z 156.655,A -85,B 0,C 180,E1 -12299.687,E2 -12299.687} C_VEL
LIN {X 0,Y 375.967,Z 156.849,A -85,B 0,C 180,E1 -12301.25,E2 -12301.25} C_VEL
LIN {X 0,Y 378.854,Z 170.961,A -85,B 0,C 180,E1 -12304.744,E2 -12304.744} C_VEL
LIN {X 0,Y 379.267,Z 176.081,A -85,B 0,C 180,E1 -12305.941,E2 -12305.941} C_VEL
LIN {X 0,Y 378.125,Z 190.037,A -85,B 0,C 180,E1 -12309.041,E2 -12309.041} C_VEL
LIN {X 0,Y 382.891,Z 221.036,A -85,B 0,C 180,E1 -12309.933,E2 -12309.933} C_VEL
LIN {X 0,Y 381.634,Z 298.999,A -85,B 0,C 180,E1 -12311.478,E2 -12311.478} C_VEL
LIN {X 0,Y 381.028,Z 312.653,A -85,B 0,C 180,E1 -12311.969,E2 -12311.969} C_VEL
LIN {X 0,Y 380.242,Z 325.515,A -85,B 0,C 180,E1 -12312.66,E2 -12312.66} C_VEL
LIN {X 0,Y 379.238,Z 338.068,A -85,B 0,C 180,E1 -12313.584,E2 -12313.584} C_VEL
LIN {X 0,Y 378.288,Z 349.287,A -85,B 0,C 180,E1 -12314.648,E2 -12314.648} C_VEL
LIN {X 0,Y 377.546,Z 358.823,A -85,B 0,C 180,E1 -12315.78,E2 -12315.78} C_VEL
LIN {X 0,Y 376.747,Z 367.69,A -85,B 0,C 180,E1 -12317.064,E2 -12317.064} C_VEL
LIN {X 0,Y 375.848,Z 376.724,A -85,B 0,C 180,E1 -12318.677,E2 -12318.677} C_VEL
LIN {X 0,Y 375.267,Z 383.998,A -85,B 0,C 180,E1 -12320.296,E2 -12320.296} C_VEL
LIN {X 0,Y 374.88,Z 389.796,A -85,B 0,C 180,E1 -12321.917,E2 -12321.917} C_VEL
LIN {X 0,Y 374.586,Z 395.26,A -85,B 0,C 180,E1 -12323.929,E2 -12323.929} C_VEL
LIN {X 0,Y 374.549,Z 398.704,A -85,B 0,C 180,E1 -12325.696,E2 -12325.696} C_VEL
LIN {X 0,Y 374.461,Z 400.238,A -85,B 0,C 180,E1 -12326.772,E2 -12326.772} C_VEL
LIN {X 0,Y 374.46,Z 401.313,A -85,B 0,C 180,E1 -12327.849,E2 -12327.849} C_VEL
LIN {X 0,Y 374.518,Z 401.987,A -85,B 0,C 180,E1 -12328.925,E2 -12328.925} C_VEL
LIN {X 0,Y 374.555,Z 402.268,A -85,B 0,C 180,E1 -12330,E2 -12330} C_VEL
LIN {X 0,Y 374.503,Z 402.151,A -85,B 0,C 180,E1 -12331.075,E2 -12331.075} C_VEL
LIN {X 0,Y 374.457,Z 401.596,A -85,B 0,C 180,E1 -12332.151,E2 -12332.151} C_VEL
LIN {X 0,Y 374.527,Z 399.289,A -85,B 0,C 180,E1 -12334.305,E2 -12334.305} C_VEL
LIN {X 0,Y 374.565,Z 396.199,A -85,B 0,C 180,E1 -12336.041,E2 -12336.041} C_VEL
LIN {X 0,Y 374.797,Z 392.552,A -85,B 0,C 180,E1 -12337.543,E2 -12337.543} C_VEL
LIN {X 0,Y 375.191,Z 387.54,A -85,B 0,C 180,E1 -12339.162,E2 -12339.162} C_VEL
LIN {X 0,Y 375.738,Z 381.248,A -85,B 0,C 180,E1 -12340.781,E2 -12340.781} C_VEL
LIN {X 0,Y 376.573,Z 373.398,A -85,B 0,C 180,E1 -12342.394,E2 -12342.394} C_VEL
LIN {X 0,Y 377.559,Z 363.6,A -85,B 0,C 180,E1 -12344.004,E2 -12344.004} C_VEL
LIN {X 0,Y 378.567,Z 353.467,A -85,B 0,C 180,E1 -12345.34,E2 -12345.34} C_VEL
LIN {X 0,Y 379.653,Z 342.011,A -85,B 0,C 180,E1 -12346.536,E2 -12346.536} C_VEL
LIN {X 0,Y 380.692,Z 330.792,A -85,B 0,C 180,E1 -12347.457,E2 -12347.457} C_VEL
LIN {X 0,Y 381.732,Z 318.219,A -85,B 0,C 180,E1 -12348.239,E2 -12348.239} C_VEL
LIN {X 0,Y 382.379,Z 306.666,A -85,B 0,C 180,E1 -12348.763,E2 -12348.763} C_VEL
LIN {X 0,Y 382.895,Z 293.331,A -85,B 0,C 180,E1 -12349.153,E2 -12349.153} C_VEL
LIN {X 0,Y 384.062,Z 220.6,A -85,B 0,C 180,E1 -12350.595,E2 -12350.595} C_VEL
LIN {X 0,Y 380.12,Z 196.628,A -85,B 0,C 180,E1 -12351.35,E2 -12351.35} C_VEL
LIN {X 0,Y 378.631,Z 189.148,A -85,B 0,C 180,E1 -12351.631,E2 -12351.631} C_VEL
LIN {X 0,Y 379.776,Z 176.407,A -85,B 0,C 180,E1 -12354.454,E2 -12354.454} C_VEL
LIN {X 0,Y 378.751,Z 169.419,A -85,B 0,C 180,E1 -12356.149,E2 -12356.149} C_VEL
LIN {X 0,Y 376.27,Z 158.05,A -85,B 0,C 180,E1 -12359.054,E2 -12359.054} C_VEL
LIN {X 0,Y 375.933,Z 156.665,A -85,B 0,C 180,E1 -12359.466,E2 -12359.466} C_VEL
LIN {X 0,Y 375.948,Z 156.661,A -85,B 0,C 180,E1 -12362.829,E2 -12362.829} C_VEL
LIN {X 0,Y 375.949,Z 156.658,A -85,B 0,C 180,E1 -12365.417,E2 -12365.417} C_VEL
LIN {X 0,Y 375.933,Z 156.656,A -85,B 0,C 180,E1 -12368.262,E2 -12368.262} C_VEL
LIN {X 0,Y 375.914,Z 156.659,A -85,B 0,C 180,E1 -12371.597,E2 -12371.597} C_VEL
LIN {X 0,Y 375.922,Z 156.659,A -85,B 0,C 180,E1 -12374.73,E2 -12374.73} C_VEL
LIN {X 0,Y 375.909,Z 156.659,A -85,B 0,C 180,E1 -12377.696,E2 -12377.696} C_VEL
LIN {X 0,Y 375.934,Z 156.653,A -85,B 0,C 180,E1 -12380.534,E2 -12380.534} C_VEL
LIN {X 0,Y 375.958,Z 156.649,A -85,B 0,C 180,E1 -12383.497,E2 -12383.497} C_VEL
LIN {X 0,Y 375.959,Z 156.651,A -85,B 0,C 180,E1 -12385.888,E2 -12385.888} C_VEL
LIN {X 0,Y 375.961,Z 156.65,A -85,B 0,C 180,E1 -12389.687,E2 -12389.687} C_VEL
LIN {X 0,Y 375.918,Z 156.654,A -85,B 0,C 180,E1 -12392.135,E2 -12392.135} C_VEL
LIN {X 0,Y 375.936,Z 156.651,A -85,B 0,C 180,E1 -12394.534,E2 -12394.534} C_VEL
LIN {X 0,Y 375.97,Z 156.653,A -85,B 0,C 180,E1 -12396.887,E2 -12396.887} C_VEL
LIN {X 0,Y 375.961,Z 156.646,A -85,B 0,C 180,E1 -12400.337,E2 -12400.337} C_VEL
LIN {X 0,Y 375.957,Z 156.648,A -85,B 0,C 180,E1 -12403.716,E2 -12403.716} C_VEL
LIN {X 0,Y 376.079,Z 156.636,A -85,B 0,C 180,E1 -12407.041,E2 -12407.041} C_VEL
LIN {X 0,Y 376.11,Z 156.631,A -85,B 0,C 180,E1 -12410.318,E2 -12410.318} C_VEL
LIN {X 0,Y 376.195,Z 156.613,A -85,B 0,C 180,E1 -12413.564,E2 -12413.564} C_VEL
LIN {X 0,Y 376.336,Z 156.598,A -85,B 0,C 180,E1 -12417.86,E2 -12417.86} C_VEL
LIN {X 0,Y 376.336,Z 156.601,A -85,B 0,C 180,E1 -12422.141,E2 -12422.141} C_VEL
LIN {X 0,Y 376.196,Z 156.622,A -85,B 0,C 180,E1 -12426.443,E2 -12426.443} C_VEL
LIN {X 0,Y 376.111,Z 156.631,A -85,B 0,C 180,E1 -12429.682,E2 -12429.682} C_VEL
LIN {X 0,Y 376.094,Z 156.637,A -85,B 0,C 180,E1 -12433.657,E2 -12433.657} C_VEL
LIN {X 0,Y 375.986,Z 156.652,A -85,B 0,C 180,E1 -12437.577,E2 -12437.577} C_VEL
LIN {X 0,Y 375.982,Z 156.649,A -85,B 0,C 180,E1 -12440.832,E2 -12440.832} C_VEL
LIN {X 0,Y 375.939,Z 156.658,A -85,B 0,C 180,E1 -12444.285,E2 -12444.285} C_VEL
LIN {X 0,Y 375.915,Z 156.662,A -85,B 0,C 180,E1 -12446.66,E2 -12446.66} C_VEL
LIN {X 0,Y 375.916,Z 156.661,A -85,B 0,C 180,E1 -12449.084,E2 -12449.084} C_VEL
LIN {X 0,Y 375.967,Z 156.717,A -85,B 0,C 180,E1 -12452.594,E2 -12452.594} C_VEL
LIN {X 0,Y 378.253,Z 167.414,A -85,B 0,C 180,E1 -12455.495,E2 -12455.495} C_VEL
LIN {X 0,Y 378.996,Z 171.347,A -85,B 0,C 180,E1 -12456.476,E2 -12456.476} C_VEL
LIN {X 0,Y 381.427,Z 180.448,A -85,B 0,C 180,E1 -12456.831,E2 -12456.831} C_VEL
LIN {X 0,Y 384.628,Z 196.293,A -85,B 0,C 180,E1 -12457.372,E2 -12457.372} C_VEL
LIN {X 0,Y 382.937,Z 279.228,A -85,B 0,C 180,E1 -12459.028,E2 -12459.028} C_VEL
LIN {X 0,Y 382.364,Z 292.784,A -85,B 0,C 180,E1 -12459.522,E2 -12459.522} C_VEL
LIN {X 0,Y 381.682,Z 305.461,A -85,B 0,C 180,E1 -12460.212,E2 -12460.212} C_VEL
LIN {X 0,Y 380.751,Z 317.552,A -85,B 0,C 180,E1 -12461.103,E2 -12461.103} C_VEL
LIN {X 0,Y 379.797,Z 328.217,A -85,B 0,C 180,E1 -12462.108,E2 -12462.108} C_VEL
LIN {X 0,Y 378.71,Z 338.887,A -85,B 0,C 180,E1 -12463.365,E2 -12463.365} C_VEL
LIN {X 0,Y 377.711,Z 348.648,A -85,B 0,C 180,E1 -12464.815,E2 -12464.815} C_VEL
LIN {X 0,Y 376.829,Z 357.078,A -85,B 0,C 180,E1 -12466.364,E2 -12466.364} C_VEL
LIN {X 0,Y 376.13,Z 363.124,A -85,B 0,C 180,E1 -12467.727,E2 -12467.727} C_VEL
LIN {X 0,Y 375.596,Z 368.113,A -85,B 0,C 180,E1 -12469.087,E2 -12469.087} C_VEL
LIN {X 0,Y 375.201,Z 372.203,A -85,B 0,C 180,E1 -12470.441,E2 -12470.441} C_VEL
LIN {X 0,Y 374.908,Z 375.803,A -85,B 0,C 180,E1 -12471.937,E2 -12471.937} C_VEL
LIN {X 0,Y 374.574,Z 379.005,A -85,B 0,C 180,E1 -12473.784,E2 -12473.784} C_VEL
LIN {X 0,Y 374.309,Z 381.036,A -85,B 0,C 180,E1 -12475.717,E2 -12475.717} C_VEL
LIN {X 0,Y 374.266,Z 381.781,A -85,B 0,C 180,E1 -12477.674,E2 -12477.674} C_VEL
LIN {X 0,Y 374.325,Z 381.126,A -85,B 0,C 180,E1 -12479.73,E2 -12479.73} C_VEL
LIN {X 0,Y 374.403,Z 380.209,A -85,B 0,C 180,E1 -12480.787,E2 -12480.787} C_VEL
LIN {X 0,Y 374.615,Z 377.664,A -85,B 0,C 180,E1 -12482.636,E2 -12482.636} C_VEL
LIN {X 0,Y 374.896,Z 373.905,A -85,B 0,C 180,E1 -12484.458,E2 -12484.458} C_VEL
LIN {X 0,Y 375.272,Z 369.147,A -85,B 0,C 180,E1 -12486.158,E2 -12486.158} C_VEL
LIN {X 0,Y 375.813,Z 362.248,A -85,B 0,C 180,E1 -12488.036,E2 -12488.036} C_VEL
LIN {X 0,Y 376.454,Z 355.45,A -85,B 0,C 180,E1 -12489.51,E2 -12489.51} C_VEL
LIN {X 0,Y 377.254,Z 347.184,A -85,B 0,C 180,E1 -12490.973,E2 -12490.973} C_VEL
LIN {X 0,Y 378.055,Z 338.167,A -85,B 0,C 180,E1 -12492.277,E2 -12492.277} C_VEL
LIN {X 0,Y 378.939,Z 328.314,A -85,B 0,C 180,E1 -12493.432,E2 -12493.432} C_VEL
LIN {X 0,Y 379.844,Z 316.936,A -85,B 0,C 180,E1 -12494.5,E2 -12494.5} C_VEL
LIN {X 0,Y 380.564,Z 305.302,A -85,B 0,C 180,E1 -12495.358,E2 -12495.358} C_VEL
LIN {X 0,Y 381.213,Z 293.026,A -85,B 0,C 180,E1 -12496.031,E2 -12496.031} C_VEL
LIN {X 0,Y 381.796,Z 279.019,A -85,B 0,C 180,E1 -12496.544,E2 -12496.544} C_VEL
LIN {X 0,Y 382.849,Z 218.754,A -85,B 0,C 180,E1 -12497.742,E2 -12497.742} C_VEL
LIN {X 0,Y 383.164,Z 194.65,A -85,B 0,C 180,E1 -12498.218,E2 -12498.218} C_VEL
LIN {X 0,Y 378.5,Z 170.589,A -85,B 0,C 180,E1 -12498.986,E2 -12498.986} C_VEL
LIN {X 0,Y 377.363,Z 163.117,A -85,B 0,C 180,E1 -12500.945,E2 -12500.945} C_VEL
LIN {X 0,Y 376.174,Z 156.626,A -85,B 0,C 180,E1 -12502.755,E2 -12502.755} C_VEL
LIN {X 0,Y 376.017,Z 156.643,A -85,B 0,C 180,E1 -12505.712,E2 -12505.712} C_VEL
LIN {X 0,Y 376.351,Z 156.603,A -85,B 0,C 180,E1 -12507.86,E2 -12507.86} C_VEL
LIN {X 0,Y 376.279,Z 156.61,A -85,B 0,C 180,E1 -12511.435,E2 -12511.435} C_VEL
LIN {X 0,Y 375.628,Z 156.698,A -85,B 0,C 180,E1 -12512.327,E2 -12512.327} C_VEL
LIN {X 0,Y 372.71,Z 157.057,A -85,B 0,C 180,E1 -12513.775,E2 -12513.775} C_VEL
LIN {X 0,Y 370.238,Z 157.364,A -85,B 0,C 180,E1 -12514.946,E2 -12514.946} C_VEL
LIN {X 0,Y 369.201,Z 157.495,A -85,B 0,C 180,E1 -12515.853,E2 -12515.853} C_VEL
LIN {X 0,Y 369.131,Z 157.501,A -85,B 0,C 180,E1 -12516.16,E2 -12516.16} C_VEL
LIN {X 0,Y 369.093,Z 157.507,A -85,B 0,C 180,E1 -12518.762,E2 -12518.762} C_VEL
LIN {X 0,Y 369.008,Z 157.523,A -85,B 0,C 180,E1 -12522.093,E2 -12522.093} C_VEL
LIN {X 0,Y 368.993,Z 157.521,A -85,B 0,C 180,E1 -12524.336,E2 -12524.336} C_VEL
LIN {X 0,Y 368.979,Z 157.524,A -85,B 0,C 180,E1 -12527.757,E2 -12527.757} C_VEL
LIN {X 0,Y 368.912,Z 157.529,A -85,B 0,C 180,E1 -12531.221,E2 -12531.221} C_VEL
LIN {X 0,Y 368.913,Z 157.534,A -85,B 0,C 180,E1 -12533.875,E2 -12533.875} C_VEL
LIN {X 0,Y 368.867,Z 157.535,A -85,B 0,C 180,E1 -12537.211,E2 -12537.211} C_VEL
LIN {X 0,Y 368.897,Z 157.536,A -85,B 0,C 180,E1 -12539.692,E2 -12539.692} C_VEL
LIN {X 0,Y 368.898,Z 157.531,A -85,B 0,C 180,E1 -12543.043,E2 -12543.043} C_VEL
LIN {X 0,Y 368.918,Z 157.528,A -85,B 0,C 180,E1 -12546.197,E2 -12546.197} C_VEL
LIN {X 0,Y 368.876,Z 157.534,A -85,B 0,C 180,E1 -12548.957,E2 -12548.957} C_VEL
LIN {X 0,Y 368.872,Z 157.534,A -85,B 0,C 180,E1 -12552.007,E2 -12552.007} C_VEL
LIN {X 0,Y 368.878,Z 157.538,A -85,B 0,C 180,E1 -12555.175,E2 -12555.175} C_VEL
LIN {X 0,Y 368.871,Z 157.533,A -85,B 0,C 180,E1 -12558.176,E2 -12558.176} C_VEL
LIN {X 0,Y 368.88,Z 157.536,A -85,B 0,C 180,E1 -12561.366,E2 -12561.366} C_VEL
LIN {X 0,Y 368.934,Z 157.531,A -85,B 0,C 180,E1 -12565.146,E2 -12565.146} C_VEL
LIN {X 0,Y 368.915,Z 157.533,A -85,B 0,C 180,E1 -12569.045,E2 -12569.045} C_VEL
LIN {X 0,Y 368.915,Z 157.529,A -85,B 0,C 180,E1 -12571.558,E2 -12571.558} C_VEL
LIN {X 0,Y 368.926,Z 157.529,A -85,B 0,C 180,E1 -12575.222,E2 -12575.222} C_VEL
LIN {X 0,Y 368.923,Z 157.53,A -85,B 0,C 180,E1 -12578.981,E2 -12578.981} C_VEL
LIN {X 0,Y 368.956,Z 157.525,A -85,B 0,C 180,E1 -12582.255,E2 -12582.255} C_VEL
LIN {X 0,Y 369.041,Z 157.515,A -85,B 0,C 180,E1 -12586.228,E2 -12586.228} C_VEL
LIN {X 0,Y 369.065,Z 157.512,A -85,B 0,C 180,E1 -12590.132,E2 -12590.132} C_VEL
LIN {X 0,Y 369.162,Z 157.497,A -85,B 0,C 180,E1 -12593.441,E2 -12593.441} C_VEL
LIN {X 0,Y 369.305,Z 157.481,A -85,B 0,C 180,E1 -12597.819,E2 -12597.819} C_VEL
LIN {X 0,Y 369.304,Z 157.485,A -85,B 0,C 180,E1 -12602.181,E2 -12602.181} C_VEL
LIN {X 0,Y 369.16,Z 157.499,A -85,B 0,C 180,E1 -12606.559,E2 -12606.559} C_VEL
LIN {X 0,Y 369.061,Z 157.515,A -85,B 0,C 180,E1 -12609.868,E2 -12609.868} C_VEL
LIN {X 0,Y 369.004,Z 157.522,A -85,B 0,C 180,E1 -12613.749,E2 -12613.749} C_VEL
LIN {X 0,Y 368.939,Z 157.531,A -85,B 0,C 180,E1 -12617.745,E2 -12617.745} C_VEL
LIN {X 0,Y 368.911,Z 157.53,A -85,B 0,C 180,E1 -12621.221,E2 -12621.221} C_VEL
LIN {X 0,Y 368.91,Z 157.532,A -85,B 0,C 180,E1 -12623.873,E2 -12623.873} C_VEL
LIN {X 0,Y 368.858,Z 157.538,A -85,B 0,C 180,E1 -12627.212,E2 -12627.212} C_VEL
LIN {X 0,Y 368.893,Z 157.534,A -85,B 0,C 180,E1 -12629.692,E2 -12629.692} C_VEL
LIN {X 0,Y 368.897,Z 157.533,A -85,B 0,C 180,E1 -12633.042,E2 -12633.042} C_VEL
LIN {X 0,Y 368.912,Z 157.528,A -85,B 0,C 180,E1 -12636.197,E2 -12636.197} C_VEL
LIN {X 0,Y 368.875,Z 157.536,A -85,B 0,C 180,E1 -12638.957,E2 -12638.957} C_VEL
LIN {X 0,Y 368.86,Z 157.535,A -85,B 0,C 180,E1 -12642.005,E2 -12642.005} C_VEL
LIN {X 0,Y 368.876,Z 157.538,A -85,B 0,C 180,E1 -12645.175,E2 -12645.175} C_VEL
LIN {X 0,Y 368.861,Z 157.535,A -85,B 0,C 180,E1 -12648.174,E2 -12648.174} C_VEL
LIN {X 0,Y 368.877,Z 157.535,A -85,B 0,C 180,E1 -12651.366,E2 -12651.366} C_VEL
LIN {X 0,Y 368.931,Z 157.529,A -85,B 0,C 180,E1 -12655.146,E2 -12655.146} C_VEL
LIN {X 0,Y 368.897,Z 157.535,A -85,B 0,C 180,E1 -12659.043,E2 -12659.043} C_VEL
LIN {X 0,Y 368.939,Z 157.644,A -85,B 0,C 180,E1 -12660.936,E2 -12660.936} C_VEL
LIN {X 0,Y 371.967,Z 172.564,A -85,B 0,C 180,E1 -12664.703,E2 -12664.703} C_VEL
LIN {X 0,Y 372.333,Z 177.003,A -85,B 0,C 180,E1 -12665.761,E2 -12665.761} C_VEL
LIN {X 0,Y 371.203,Z 189.882,A -85,B 0,C 180,E1 -12668.675,E2 -12668.675} C_VEL
LIN {X 0,Y 376.108,Z 222.14,A -85,B 0,C 180,E1 -12669.619,E2 -12669.619} C_VEL
LIN {X 0,Y 374.833,Z 298.689,A -85,B 0,C 180,E1 -12671.165,E2 -12671.165} C_VEL
LIN {X 0,Y 374.214,Z 312.378,A -85,B 0,C 180,E1 -12671.665,E2 -12671.665} C_VEL
LIN {X 0,Y 373.455,Z 324.759,A -85,B 0,C 180,E1 -12672.335,E2 -12672.335} C_VEL
LIN {X 0,Y 372.375,Z 337.431,A -85,B 0,C 180,E1 -12673.272,E2 -12673.272} C_VEL
LIN {X 0,Y 371.401,Z 348.734,A -85,B 0,C 180,E1 -12674.356,E2 -12674.356} C_VEL
LIN {X 0,Y 370.584,Z 358.772,A -85,B 0,C 180,E1 -12675.566,E2 -12675.566} C_VEL
LIN {X 0,Y 369.777,Z 367.273,A -85,B 0,C 180,E1 -12676.816,E2 -12676.816} C_VEL
LIN {X 0,Y 368.831,Z 376.349,A -85,B 0,C 180,E1 -12678.459,E2 -12678.459} C_VEL
LIN {X 0,Y 368.226,Z 383.661,A -85,B 0,C 180,E1 -12680.109,E2 -12680.109} C_VEL
LIN {X 0,Y 367.838,Z 389.499,A -85,B 0,C 180,E1 -12681.761,E2 -12681.761} C_VEL
LIN {X 0,Y 367.563,Z 394.079,A -85,B 0,C 180,E1 -12683.412,E2 -12683.412} C_VEL
LIN {X 0,Y 367.463,Z 396.486,A -85,B 0,C 180,E1 -12684.512,E2 -12684.512} C_VEL
LIN {X 0,Y 367.454,Z 398.457,A -85,B 0,C 180,E1 -12685.612,E2 -12685.612} C_VEL
LIN {X 0,Y 367.379,Z 400.004,A -85,B 0,C 180,E1 -12686.71,E2 -12686.71} C_VEL
LIN {X 0,Y 367.361,Z 401.095,A -85,B 0,C 180,E1 -12687.807,E2 -12687.807} C_VEL
LIN {X 0,Y 367.418,Z 401.778,A -85,B 0,C 180,E1 -12688.904,E2 -12688.904} C_VEL
LIN {X 0,Y 367.457,Z 402.068,A -85,B 0,C 180,E1 -12690,E2 -12690} C_VEL
LIN {X 0,Y 367.403,Z 401.963,A -85,B 0,C 180,E1 -12691.096,E2 -12691.096} C_VEL
LIN {X 0,Y 367.358,Z 401.422,A -85,B 0,C 180,E1 -12692.193,E2 -12692.193} C_VEL
LIN {X 0,Y 367.377,Z 400.477,A -85,B 0,C 180,E1 -12693.29,E2 -12693.29} C_VEL
LIN {X 0,Y 367.435,Z 399.134,A -85,B 0,C 180,E1 -12694.388,E2 -12694.388} C_VEL
LIN {X 0,Y 367.473,Z 396.364,A -85,B 0,C 180,E1 -12696.005,E2 -12696.005} C_VEL
LIN {X 0,Y 367.722,Z 392.433,A -85,B 0,C 180,E1 -12697.689,E2 -12697.689} C_VEL
LIN {X 0,Y 368.14,Z 387.44,A -85,B 0,C 180,E1 -12699.339,E2 -12699.339} C_VEL
LIN {X 0,Y 368.719,Z 381.169,A -85,B 0,C 180,E1 -12700.988,E2 -12700.988} C_VEL
LIN {X 0,Y 369.629,Z 373.357,A -85,B 0,C 180,E1 -12702.63,E2 -12702.63} C_VEL
LIN {X 0,Y 370.507,Z 365.382,A -85,B 0,C 180,E1 -12703.996,E2 -12703.996} C_VEL
LIN {X 0,Y 371.475,Z 355.667,A -85,B 0,C 180,E1 -12705.359,E2 -12705.359} C_VEL
LIN {X 0,Y 372.599,Z 344.906,A -85,B 0,C 180,E1 -12706.576,E2 -12706.576} C_VEL
LIN {X 0,Y 373.608,Z 334.499,A -85,B 0,C 180,E1 -12707.517,E2 -12707.517} C_VEL
LIN {X 0,Y 374.674,Z 323.151,A -85,B 0,C 180,E1 -12708.312,E2 -12708.312} C_VEL
LIN {X 0,Y 375.455,Z 310.483,A -85,B 0,C 180,E1 -12708.98,E2 -12708.98} C_VEL
LIN {X 0,Y 376.216,Z 297.383,A -85,B 0,C 180,E1 -12709.436,E2 -12709.436} C_VEL
LIN {X 0,Y 377.497,Z 221.492,A -85,B 0,C 180,E1 -12710.988,E2 -12710.988} C_VEL
LIN {X 0,Y 373.787,Z 198.671,A -85,B 0,C 180,E1 -12711.724,E2 -12711.724} C_VEL
LIN {X 0,Y 371.835,Z 188.919,A -85,B 0,C 180,E1 -12712.096,E2 -12712.096} C_VEL
LIN {X 0,Y 372.877,Z 178.29,A -85,B 0,C 180,E1 -12714.498,E2 -12714.498} C_VEL
LIN {X 0,Y 372.296,Z 173.232,A -85,B 0,C 180,E1 -12715.733,E2 -12715.733} C_VEL
LIN {X 0,Y 369.63,Z 160.627,A -85,B 0,C 180,E1 -12718.999,E2 -12718.999} C_VEL
LIN {X 0,Y 368.906,Z 157.541,A -85,B 0,C 180,E1 -12719.849,E2 -12719.849} C_VEL
LIN {X 0,Y 368.896,Z 157.538,A -85,B 0,C 180,E1 -12723.539,E2 -12723.539} C_VEL
LIN {X 0,Y 368.896,Z 157.534,A -85,B 0,C 180,E1 -12726.854,E2 -12726.854} C_VEL
LIN {X 0,Y 368.885,Z 157.536,A -85,B 0,C 180,E1 -12730.374,E2 -12730.374} C_VEL
LIN {X 0,Y 368.88,Z 157.537,A -85,B 0,C 180,E1 -12733.615,E2 -12733.615} C_VEL
LIN {X 0,Y 368.885,Z 157.536,A -85,B 0,C 180,E1 -12736.696,E2 -12736.696} C_VEL
LIN {X 0,Y 368.886,Z 157.53,A -85,B 0,C 180,E1 -12739.648,E2 -12739.648} C_VEL
LIN {X 0,Y 368.896,Z 157.529,A -85,B 0,C 180,E1 -12743.146,E2 -12743.146} C_VEL
LIN {X 0,Y 368.897,Z 157.53,A -85,B 0,C 180,E1 -12746.462,E2 -12746.462} C_VEL
LIN {X 0,Y 368.898,Z 157.533,A -85,B 0,C 180,E1 -12749.044,E2 -12749.044} C_VEL
LIN {X 0,Y 368.909,Z 157.526,A -85,B 0,C 180,E1 -12751.558,E2 -12751.558} C_VEL
LIN {X 0,Y 368.921,Z 157.528,A -85,B 0,C 180,E1 -12754.014,E2 -12754.014} C_VEL
LIN {X 0,Y 368.896,Z 157.531,A -85,B 0,C 180,E1 -12757.603,E2 -12757.603} C_VEL
LIN {X 0,Y 368.902,Z 157.532,A -85,B 0,C 180,E1 -12761.103,E2 -12761.103} C_VEL
LIN {X 0,Y 368.923,Z 157.523,A -85,B 0,C 180,E1 -12764.532,E2 -12764.532} C_VEL
LIN {X 0,Y 369.026,Z 157.516,A -85,B 0,C 180,E1 -12766.789,E2 -12766.789} C_VEL
LIN {X 0,Y 369.06,Z 157.507,A -85,B 0,C 180,E1 -12770.132,E2 -12770.132} C_VEL
LIN {X 0,Y 369.127,Z 157.499,A -85,B 0,C 180,E1 -12772.341,E2 -12772.341} C_VEL
LIN {X 0,Y 369.117,Z 157.502,A -85,B 0,C 180,E1 -12774.537,E2 -12774.537} C_VEL
LIN {X 0,Y 369.299,Z 157.475,A -85,B 0,C 180,E1 -12777.819,E2 -12777.819} C_VEL
LIN {X 0,Y 369.206,Z 157.489,A -85,B 0,C 180,E1 -12781.091,E2 -12781.091} C_VEL
LIN {X 0,Y 369.299,Z 157.477,A -85,B 0,C 180,E1 -12782.181,E2 -12782.181} C_VEL
LIN {X 0,Y 369.158,Z 157.5,A -85,B 0,C 180,E1 -12786.559,E2 -12786.559} C_VEL
LIN {X 0,Y 369.062,Z 157.51,A -85,B 0,C 180,E1 -12789.869,E2 -12789.869} C_VEL
LIN {X 0,Y 369.041,Z 157.516,A -85,B 0,C 180,E1 -12793.772,E2 -12793.772} C_VEL
LIN {X 0,Y 368.957,Z 157.526,A -85,B 0,C 180,E1 -12797.745,E2 -12797.745} C_VEL
LIN {X 0,Y 368.912,Z 157.531,A -85,B 0,C 180,E1 -12801.221,E2 -12801.221} C_VEL
LIN {X 0,Y 368.914,Z 157.534,A -85,B 0,C 180,E1 -12803.875,E2 -12803.875} C_VEL
LIN {X 0,Y 368.861,Z 157.543,A -85,B 0,C 180,E1 -12807.212,E2 -12807.212} C_VEL
LIN {X 0,Y 368.896,Z 157.536,A -85,B 0,C 180,E1 -12809.692,E2 -12809.692} C_VEL
LIN {X 0,Y 368.929,Z 157.598,A -85,B 0,C 180,E1 -12812.191,E2 -12812.191} C_VEL
LIN {X 0,Y 371.202,Z 168.101,A -85,B 0,C 180,E1 -12815.107,E2 -12815.107} C_VEL
LIN {X 0,Y 371.87,Z 171.513,A -85,B 0,C 180,E1 -12815.99,E2 -12815.99} C_VEL
LIN {X 0,Y 374.378,Z 179.248,A -85,B 0,C 180,E1 -12816.335,E2 -12816.335} C_VEL
LIN {X 0,Y 378.083,Z 197.017,A -85,B 0,C 180,E1 -12816.967,E2 -12816.967} C_VEL
LIN {X 0,Y 376.344,Z 278.993,A -85,B 0,C 180,E1 -12818.63,E2 -12818.63} C_VEL
LIN {X 0,Y 375.722,Z 292.72,A -85,B 0,C 180,E1 -12819.133,E2 -12819.133} C_VEL
LIN {X 0,Y 375.086,Z 304.974,A -85,B 0,C 180,E1 -12819.805,E2 -12819.805} C_VEL
LIN {X 0,Y 374.125,Z 316.775,A -85,B 0,C 180,E1 -12820.672,E2 -12820.672} C_VEL
LIN {X 0,Y 373.088,Z 327.829,A -85,B 0,C 180,E1 -12821.717,E2 -12821.717} C_VEL
LIN {X 0,Y 372.097,Z 337.394,A -85,B 0,C 180,E1 -12822.84,E2 -12822.84} C_VEL
LIN {X 0,Y 370.969,Z 347.466,A -85,B 0,C 180,E1 -12824.301,E2 -12824.301} C_VEL
LIN {X 0,Y 370.018,Z 356.012,A -85,B 0,C 180,E1 -12825.854,E2 -12825.854} C_VEL
LIN {X 0,Y 369.204,Z 363.021,A -85,B 0,C 180,E1 -12827.425,E2 -12827.425} C_VEL
LIN {X 0,Y 368.494,Z 369.39,A -85,B 0,C 180,E1 -12829.214,E2 -12829.214} C_VEL
LIN {X 0,Y 368.033,Z 374.113,A -85,B 0,C 180,E1 -12830.937,E2 -12830.937} C_VEL
LIN {X 0,Y 367.74,Z 376.983,A -85,B 0,C 180,E1 -12832.297,E2 -12832.297} C_VEL
LIN {X 0,Y 367.513,Z 379.167,A -85,B 0,C 180,E1 -12833.642,E2 -12833.642} C_VEL
LIN {X 0,Y 367.247,Z 381.045,A -85,B 0,C 180,E1 -12835.376,E2 -12835.376} C_VEL
LIN {X 0,Y 367.166,Z 381.972,A -85,B 0,C 180,E1 -12837.591,E2 -12837.591} C_VEL
LIN {X 0,Y 367.208,Z 381.497,A -85,B 0,C 180,E1 -12839.458,E2 -12839.458} C_VEL
LIN {X 0,Y 367.397,Z 379.435,A -85,B 0,C 180,E1 -12841.636,E2 -12841.636} C_VEL
LIN {X 0,Y 367.641,Z 376.752,A -85,B 0,C 180,E1 -12843.305,E2 -12843.305} C_VEL
LIN {X 0,Y 367.993,Z 372.548,A -85,B 0,C 180,E1 -12845.155,E2 -12845.155} C_VEL
LIN {X 0,Y 368.384,Z 367.031,A -85,B 0,C 180,E1 -12846.977,E2 -12846.977} C_VEL
LIN {X 0,Y 369.039,Z 359.915,A -85,B 0,C 180,E1 -12848.787,E2 -12848.787} C_VEL
LIN {X 0,Y 369.755,Z 352.567,A -85,B 0,C 180,E1 -12850.283,E2 -12850.283} C_VEL
LIN {X 0,Y 370.717,Z 342.969,A -85,B 0,C 180,E1 -12851.864,E2 -12851.864} C_VEL
LIN {X 0,Y 371.569,Z 333.732,A -85,B 0,C 180,E1 -12853.093,E2 -12853.093} C_VEL
LIN {X 0,Y 372.613,Z 322.051,A -85,B 0,C 180,E1 -12854.332,E2 -12854.332} C_VEL
LIN {X 0,Y 373.457,Z 309.809,A -85,B 0,C 180,E1 -12855.352,E2 -12855.352} C_VEL
LIN {X 0,Y 374.173,Z 296.968,A -85,B 0,C 180,E1 -12856.144,E2 -12856.144} C_VEL
LIN {X 0,Y 374.827,Z 283.822,A -85,B 0,C 180,E1 -12856.711,E2 -12856.711} C_VEL
LIN {X 0,Y 375.22,Z 270.111,A -85,B 0,C 180,E1 -12857.065,E2 -12857.065} C_VEL
LIN {X 0,Y 376.398,Z 195.388,A -85,B 0,C 180,E1 -12858.549,E2 -12858.549} C_VEL
LIN {X 0,Y 371.53,Z 170.861,A -85,B 0,C 180,E1 -12859.337,E2 -12859.337} C_VEL
LIN {X 0,Y 369.566,Z 159.713,A -85,B 0,C 180,E1 -12862.35,E2 -12862.35} C_VEL
LIN {X 0,Y 369.15,Z 157.502,A -85,B 0,C 180,E1 -12862.994,E2 -12862.994} C_VEL
LIN {X 0,Y 369.115,Z 157.506,A -85,B 0,C 180,E1 -12866.725,E2 -12866.725} C_VEL
LIN {X 0,Y 369.316,Z 157.479,A -85,B 0,C 180,E1 -12867.819,E2 -12867.819} C_VEL
LIN {X 0,Y 369.245,Z 157.487,A -85,B 0,C 180,E1 -12871.442,E2 -12871.442} C_VEL
LIN {X 0,Y 369.082,Z 157.507,A -85,B 0,C 180,E1 -12873.275,E2 -12873.275} C_VEL
LIN {X 0,Y 369.131,Z 157.501,A -85,B 0,C 180,E1 -12876.16,E2 -12876.16} C_VEL
LIN {X 0,Y 368.492,Z 157.584,A -85,B 0,C 180,E1 -12877.071,E2 -12877.071} C_VEL
LIN {X 0,Y 365.6,Z 157.945,A -85,B 0,C 180,E1 -12878.55,E2 -12878.55} C_VEL
LIN {X 0,Y 363.125,Z 158.251,A -85,B 0,C 180,E1 -12879.746,E2 -12879.746} C_VEL
LIN {X 0,Y 362.06,Z 158.383,A -85,B 0,C 180,E1 -12880.673,E2 -12880.673} C_VEL
LIN {X 0,Y 361.973,Z 158.392,A -85,B 0,C 180,E1 -12880.987,E2 -12880.987} C_VEL
LIN {X 0,Y 361.982,Z 158.396,A -85,B 0,C 180,E1 -12883.887,E2 -12883.887} C_VEL
LIN {X 0,Y 361.913,Z 158.405,A -85,B 0,C 180,E1 -12888.102,E2 -12888.102} C_VEL
LIN {X 0,Y 361.856,Z 158.411,A -85,B 0,C 180,E1 -12891.655,E2 -12891.655} C_VEL
LIN {X 0,Y 361.863,Z 158.408,A -85,B 0,C 180,E1 -12895.295,E2 -12895.295} C_VEL
LIN {X 0,Y 361.857,Z 158.408,A -85,B 0,C 180,E1 -12899.074,E2 -12899.074} C_VEL
LIN {X 0,Y 361.85,Z 158.409,A -85,B 0,C 180,E1 -12902.945,E2 -12902.945} C_VEL
LIN {X 0,Y 361.869,Z 158.411,A -85,B 0,C 180,E1 -12905.637,E2 -12905.637} C_VEL
LIN {X 0,Y 361.828,Z 158.413,A -85,B 0,C 180,E1 -12909.018,E2 -12909.018} C_VEL
LIN {X 0,Y 361.835,Z 158.411,A -85,B 0,C 180,E1 -12912.829,E2 -12912.829} C_VEL
LIN {X 0,Y 361.816,Z 158.413,A -85,B 0,C 180,E1 -12915.948,E2 -12915.948} C_VEL
LIN {X 0,Y 361.815,Z 158.418,A -85,B 0,C 180,E1 -12919.249,E2 -12919.249} C_VEL
LIN {X 0,Y 361.865,Z 158.411,A -85,B 0,C 180,E1 -12922.982,E2 -12922.982} C_VEL
LIN {X 0,Y 361.86,Z 158.409,A -85,B 0,C 180,E1 -12926.631,E2 -12926.631} C_VEL
LIN {X 0,Y 361.859,Z 158.407,A -85,B 0,C 180,E1 -12929.67,E2 -12929.67} C_VEL
LIN {X 0,Y 361.866,Z 158.407,A -85,B 0,C 180,E1 -12933.468,E2 -12933.468} C_VEL
LIN {X 0,Y 361.867,Z 158.408,A -85,B 0,C 180,E1 -12937.143,E2 -12937.143} C_VEL
LIN {X 0,Y 361.865,Z 158.412,A -85,B 0,C 180,E1 -12940.721,E2 -12940.721} C_VEL
LIN {X 0,Y 361.898,Z 158.405,A -85,B 0,C 180,E1 -12944.224,E2 -12944.224} C_VEL
LIN {X 0,Y 362.003,Z 158.395,A -85,B 0,C 180,E1 -12946.528,E2 -12946.528} C_VEL
LIN {X 0,Y 362.002,Z 158.391,A -85,B 0,C 180,E1 -12949.937,E2 -12949.937} C_VEL
LIN {X 0,Y 362.126,Z 158.374,A -85,B 0,C 180,E1 -12953.313,E2 -12953.313} C_VEL
LIN {X 0,Y 362.268,Z 158.358,A -85,B 0,C 180,E1 -12957.776,E2 -12957.776} C_VEL
LIN {X 0,Y 362.178,Z 158.367,A -85,B 0,C 180,E1 -12961.112,E2 -12961.112} C_VEL
LIN {X 0,Y 362.267,Z 158.361,A -85,B 0,C 180,E1 -12962.224,E2 -12962.224} C_VEL
LIN {X 0,Y 362.125,Z 158.374,A -85,B 0,C 180,E1 -12966.687,E2 -12966.687} C_VEL
LIN {X 0,Y 361.997,Z 158.395,A -85,B 0,C 180,E1 -12970.063,E2 -12970.063} C_VEL
LIN {X 0,Y 361.954,Z 158.401,A -85,B 0,C 180,E1 -12973.868,E2 -12973.868} C_VEL
LIN {X 0,Y 361.898,Z 158.407,A -85,B 0,C 180,E1 -12977.903,E2 -12977.903} C_VEL
LIN {X 0,Y 361.855,Z 158.414,A -85,B 0,C 180,E1 -12981.655,E2 -12981.655} C_VEL
LIN {X 0,Y 361.854,Z 158.411,A -85,B 0,C 180,E1 -12985.296,E2 -12985.296} C_VEL
LIN {X 0,Y 361.858,Z 158.409,A -85,B 0,C 180,E1 -12989.073,E2 -12989.073} C_VEL
LIN {X 0,Y 361.849,Z 158.41,A -85,B 0,C 180,E1 -12992.945,E2 -12992.945} C_VEL
LIN {X 0,Y 361.865,Z 158.409,A -85,B 0,C 180,E1 -12995.637,E2 -12995.637} C_VEL
LIN {X 0,Y 361.827,Z 158.415,A -85,B 0,C 180,E1 -12999.018,E2 -12999.018} C_VEL
LIN {X 0,Y 361.831,Z 158.413,A -85,B 0,C 180,E1 -13002.83,E2 -13002.83} C_VEL
LIN {X 0,Y 361.815,Z 158.412,A -85,B 0,C 180,E1 -13005.947,E2 -13005.947} C_VEL
LIN {X 0,Y 361.812,Z 158.416,A -85,B 0,C 180,E1 -13009.249,E2 -13009.249} C_VEL
LIN {X 0,Y 361.862,Z 158.412,A -85,B 0,C 180,E1 -13012.981,E2 -13012.981} C_VEL
LIN {X 0,Y 361.858,Z 158.411,A -85,B 0,C 180,E1 -13016.631,E2 -13016.631} C_VEL
LIN {X 0,Y 361.884,Z 158.478,A -85,B 0,C 180,E1 -13020.623,E2 -13020.623} C_VEL
LIN {X 0,Y 364.511,Z 171.467,A -85,B 0,C 180,E1 -13023.981,E2 -13023.981} C_VEL
LIN {X 0,Y 365.372,Z 176.629,A -85,B 0,C 180,E1 -13025.268,E2 -13025.268} C_VEL
LIN {X 0,Y 364.724,Z 185.513,A -85,B 0,C 180,E1 -13027.332,E2 -13027.332} C_VEL
LIN {X 0,Y 364.316,Z 189.738,A -85,B 0,C 180,E1 -13028.302,E2 -13028.302} C_VEL
LIN {X 0,Y 369.379,Z 222.716,A -85,B 0,C 180,E1 -13029.285,E2 -13029.285} C_VEL
LIN {X 0,Y 368.052,Z 298.382,A -85,B 0,C 180,E1 -13030.84,E2 -13030.84} C_VEL
LIN {X 0,Y 367.422,Z 312.103,A -85,B 0,C 180,E1 -13031.349,E2 -13031.349} C_VEL
LIN {X 0,Y 366.636,Z 323.958,A -85,B 0,C 180,E1 -13031.995,E2 -13031.995} C_VEL
LIN {X 0,Y 365.704,Z 335.211,A -85,B 0,C 180,E1 -13032.814,E2 -13032.814} C_VEL
LIN {X 0,Y 364.624,Z 346.879,A -85,B 0,C 180,E1 -13033.914,E2 -13033.914} C_VEL
LIN {X 0,Y 363.677,Z 358.013,A -85,B 0,C 180,E1 -13035.246,E2 -13035.246} C_VEL
LIN {X 0,Y 362.805,Z 366.853,A -85,B 0,C 180,E1 -13036.558,E2 -13036.558} C_VEL
LIN {X 0,Y 361.842,Z 375.97,A -85,B 0,C 180,E1 -13038.232,E2 -13038.232} C_VEL
LIN {X 0,Y 361.205,Z 383.316,A -85,B 0,C 180,E1 -13039.915,E2 -13039.915} C_VEL
LIN {X 0,Y 360.78,Z 389.19,A -85,B 0,C 180,E1 -13041.599,E2 -13041.599} C_VEL
LIN {X 0,Y 360.497,Z 393.799,A -85,B 0,C 180,E1 -13043.283,E2 -13043.283} C_VEL
